C01894=67.036,-67.036,18.916,160.1256,-19.8741,0.0000
C01895=63.169,-70.689,18.914,159.1053,-18.7979,0.0000
C01896=59.448,-73.859,18.917,158.5547,-18.0191,0.0000
C01897=56.048,-76.685,18.976,160.0045,-17.9572,0.0000
C01898=53.950,-78.738,19.120,165.3862,-17.8366,0.0000
C01899=52.755,-80.388,19.309,171.7434,-14.7955,0.0000
C01900=51.961,-81.931,19.493,175.4363,-10.0997,0.0000
C01901=51.163,-83.502,19.627,176.4604,-6.1368,0.0000
C01902=49.917,-85.194,19.692,177.1673,-3.1412,0.0000
C01903=47.874,-87.106,19.726,178.6253,-1.1228,0.0000
C01904=45.272,-88.975,19.753,179.7684,-0.1462,0.0000
C01905=42.449,-90.515,19.780,179.9313,-0.0331,0.0000
C01906=39.659,-91.796,19.798,179.9923,-0.0034,0.0000
C01907=36.867,-92.953,19.798,179.9922,-0.0031,0.0000
C01908=33.988,-94.020,19.780,179.9280,-0.0252,0.0000
C01909=30.903,-94.927,19.753,179.7329,-0.0604,0.0000
C01910=27.741,-95.446,19.726,178.2343,-0.1783,0.0000
C01911=24.945,-95.538,19.692,175.7796,0.2187,0.0000
C01912=22.867,-95.222,19.627,173.1704,1.8493,0.0000
C01913=21.192,-94.676,19.493,169.6633,3.9762,0.0000
C01914=19.540,-94.146,19.309,163.8609,4.8105,0.0000
C01915=17.528,-93.824,19.120,157.6135,2.4711,0.0000
C01916=14.592,-93.857,18.976,154.0583,-1.6112,0.0000
C01917=10.190,-94.262,18.917,153.0799,-2.7339,0.0000
C01918=5.317,-94.652,18.914,152.9496,-1.6759,0.0000
C01919=0.000,-94.804,18.916,152.9230,0.0002,0.0000
C01920=0.000,-94.804,18.916,152.9230,0.0002,0.0000
C01921=-5.317,-94.652,18.914,152.9496,1.6756,0.0000
C01922=-10.190,-94.262,18.917,153.0799,2.7335,0.0000
C01923=-14.592,-93.857,18.976,154.0584,1.6115,0.0000
C01924=-17.528,-93.824,19.120,157.6135,-2.4711,0.0000
C01925=-19.540,-94.146,19.309,163.8609,-4.8105,0.0000
C01926=-21.192,-94.676,19.493,169.6633,-3.9762,0.0000
C01927=-22.867,-95.222,19.627,173.1704,-1.8493,0.0000
C01928=-24.945,-95.538,19.692,175.7796,-0.2187,0.0000
C01929=-27.741,-95.446,19.726,178.2343,0.1783,0.0000
C01930=-30.903,-94.927,19.753,179.7329,0.0604,0.0000
C01931=-33.988,-94.020,19.780,179.9280,0.0252,0.0000
C01932=-36.867,-92.953,19.798,179.9922,0.0031,0.0000
C01933=-39.659,-91.796,19.798,179.9923,0.0034,0.0000
C01934=-42.449,-90.515,19.780,179.9313,0.0331,0.0000
C01935=-45.272,-88.975,19.753,179.7684,0.1462,0.0000
C01936=-47.874,-87.106,19.726,178.6253,1.1228,0.0000
C01937=-49.917,-85.194,19.692,177.1673,3.1412,0.0000
C01938=-51.163,-83.502,19.627,176.4604,6.1368,0.0000
C01939=-51.961,-81.931,19.493,175.4363,10.0997,0.0000
C01940=-52.755,-80.388,19.309,171.7434,14.7955,0.0000
C01941=-53.950,-78.738,19.120,165.3862,17.8366,0.0000
C01942=-56.048,-76.685,18.976,160.0047,17.9574,0.0000
C01943=-59.448,-73.859,18.917,158.5544,18.0188,0.0000
C01944=-63.169,-70.689,18.914,159.1051,18.7977,0.0000
C01945=-67.036,-67.036,18.916,160.1259,19.8744,0.0000
C01946=-70.689,-63.169,18.914,161.2021,20.8947,0.0000
C01947=-73.859,-59.448,18.917,161.9809,21.4453,0.0000
C01948=-76.685,-56.048,18.976,162.0428,19.9955,0.0000
C01949=-78.738,-53.950,19.120,162.1634,14.6138,0.0000
C01950=-80.388,-52.755,19.309,165.2045,8.2566,0.0000
C01951=-81.931,-51.961,19.493,169.9003,4.5637,0.0000
C01952=-83.502,-51.163,19.627,173.8632,3.5396,0.0000
C01953=-85.194,-49.917,19.692,176.8588,2.8327,0.0000
C01954=-87.106,-47.874,19.726,178.8772,1.3747,0.0000
C01955=-88.975,-45.272,19.753,179.8538,0.2316,0.0000
C01956=-90.515,-42.449,19.780,179.9669,0.0687,0.0000
C01957=-91.796,-39.659,19.798,179.9966,0.0077,0.0000
C01958=-92.953,-36.867,19.798,179.9969,0.0078,0.0000
C01959=-94.020,-33.988,19.780,179.9748,0.0720,0.0000
C01960=-94.927,-30.903,19.753,179.9396,0.2671,0.0000
C01961=-95.446,-27.741,19.726,179.8217,1.7657,0.0000
C01962=-95.538,-24.945,19.692,-179.7813,4.2204,0.0000
C01963=-95.222,-22.867,19.627,-178.1507,6.8296,0.0000
C01964=-94.676,-21.192,19.493,-176.0238,10.3367,0.0000
C01965=-94.146,-19.540,19.309,-175.1895,16.1391,0.0000
C01966=-93.824,-17.528,19.120,-177.5289,22.3865,0.0000
C01967=-93.857,-14.592,18.976,178.3888,25.9417,0.0000
C01968=-94.262,-10.190,18.917,177.2661,26.9201,0.0000
C01969=-94.652,-5.317,18.914,178.3241,27.0504,0.0000
C01970=-94.804,0.000,18.916,-179.9998,27.0770,0.0000
C01971=-94.652,5.317,18.914,-178.3244,27.0504,0.0000
C01972=-94.262,10.190,18.917,-177.2665,26.9201,0.0000
C01973=-93.857,14.592,18.976,-178.3885,25.9416,0.0000
C01974=-93.824,17.528,19.120,177.5289,22.3865,0.0000
C01975=-94.146,19.540,19.309,175.1895,16.1391,0.0000
C01976=-94.676,21.192,19.493,176.0238,10.3367,0.0000
C01977=-95.222,22.867,19.627,178.1507,6.8296,0.0000
C01978=-95.538,24.945,19.692,179.7813,4.2204,0.0000
C01979=-95.446,27.741,19.726,-179.8217,1.7657,0.0000
C01980=-94.927,30.903,19.753,-179.9396,0.2671,0.0000
C01981=-94.020,33.988,19.780,-179.9748,0.0720,0.0000
C01982=-92.953,36.867,19.798,-179.9969,0.0078,0.0000
C01983=-91.796,39.659,19.798,-179.9966,0.0077,0.0000
C01984=-90.515,42.449,19.780,-179.9669,0.0687,0.0000
C01985=-88.975,45.272,19.753,-179.8538,0.2316,0.0000
C01986=-87.106,47.874,19.726,-178.8772,1.3747,0.0000
C01987=-85.194,49.917,19.692,-176.8588,2.8327,0.0000
C01988=-83.502,51.163,19.627,-173.8632,3.5396,0.0000
C01989=-81.931,51.961,19.493,-169.9003,4.5637,0.0000
C01990=-80.388,52.755,19.309,-165.2045,8.2566,0.0000
C01991=-78.738,53.950,19.120,-162.1634,14.6138,0.0000
C01992=-76.685,56.048,18.976,-162.0426,19.9953,0.0000
C01993=-73.859,59.448,18.917,-161.9812,21.4456,0.0000
C01994=-70.689,63.169,18.914,-161.2023,20.8949,0.0000
C01995=-67.036,67.036,18.916,-160.1256,19.8741,0.0000
C01996=-63.169,70.689,18.914,-159.1053,18.7979,0.0000
C01997=-59.448,73.859,18.917,-158.5547,18.0191,0.0000
C01998=-56.048,76.685,18.976,-160.0045,17.9572,0.0000
C01999=-53.950,78.738,19.120,-165.3862,17.8366,0.0000
///TOOL 0
///POSTYPE ANGLE
///ANGLE
EC00000=0.0000,0.0000
EC00001=0.0000,0.0000
EC00002=3.3204,0.0000
EC00003=6.3084,0.0000
EC00004=8.9540,0.0000
EC00005=10.7765,0.0000
EC00006=12.0369,0.0000
EC00007=13.0576,0.0000
EC00008=14.0938,0.0000
EC00009=15.3967,0.0000
EC00010=17.0065,0.0000
EC00011=18.7198,0.0000
EC00012=20.3278,0.0000
EC00013=21.7902,0.0000
EC00014=23.2098,0.0000
EC00015=24.6724,0.0000
EC00016=26.2801,0.0000
EC00017=27.9935,0.0000
EC00018=29.6039,0.0000
EC00019=30.9060,0.0000
EC00020=31.9421,0.0000
EC00021=32.9632,0.0000
EC00022=34.2234,0.0000
EC00023=36.0464,0.0000
EC00024=38.6909,0.0000
EC00025=41.6796,0.0000
EC00026=45.0000,0.0000
EC00027=48.3204,0.0000
EC00028=51.3091,0.0000
EC00029=53.9536,0.0000
EC00030=55.7766,0.0000
EC00031=57.0368,0.0000
EC00032=58.0579,0.0000
EC00033=59.0940,0.0000
EC00034=60.3961,0.0000
EC00035=62.0065,0.0000
EC00036=63.7199,0.0000
EC00037=65.3276,0.0000
EC00038=66.7902,0.0000
EC00039=68.2098,0.0000
EC00040=69.6722,0.0000
EC00041=71.2802,0.0000
EC00042=72.9935,0.0000
EC00043=74.6033,0.0000
EC00044=75.9062,0.0000
EC00045=76.9424,0.0000
EC00046=77.9631,0.0000
EC00047=79.2235,0.0000
EC00048=81.0460,0.0000
EC00049=83.6916,0.0000
EC00050=86.6796,0.0000
EC00051=90.0000,0.0000
EC00052=93.3204,0.0000
EC00053=96.3084,0.0000
EC00054=98.9540,0.0000
EC00055=100.7765,0.0000
EC00056=102.0369,0.0000
EC00057=103.0576,0.0000
EC00058=104.0938,0.0000
EC00059=105.3967,0.0000
EC00060=107.0065,0.0000
EC00061=108.7198,0.0000
EC00062=110.3278,0.0000
EC00063=111.7902,0.0000
EC00064=113.2098,0.0000
EC00065=114.6724,0.0000
EC00066=116.2801,0.0000
EC00067=117.9935,0.0000
EC00068=119.6039,0.0000
EC00069=120.9060,0.0000
EC00070=121.9421,0.0000
EC00071=122.9632,0.0000
EC00072=124.2234,0.0000
EC00073=126.0464,0.0000
EC00074=128.6909,0.0000
EC00075=131.6796,0.0000
EC00076=135.0000,0.0000
EC00077=138.3204,0.0000
EC00078=141.3091,0.0000
EC00079=143.9536,0.0000
EC00080=145.7766,0.0000
EC00081=147.0368,0.0000
EC00082=148.0579,0.0000
EC00083=149.0940,0.0000
EC00084=150.3961,0.0000
EC00085=152.0065,0.0000
EC00086=153.7199,0.0000
EC00087=155.3276,0.0000
EC00088=156.7902,0.0000
EC00089=158.2098,0.0000
EC00090=159.6722,0.0000
EC00091=161.2802,0.0000
EC00092=162.9935,0.0000
EC00093=164.6033,0.0000
EC00094=165.9062,0.0000
EC00095=166.9424,0.0000
EC00096=167.9631,0.0000
EC00097=169.2235,0.0000
EC00098=171.0460,0.0000
EC00099=173.6916,0.0000
EC00100=176.6796,0.0000
EC00101=180.0000,0.0000
EC00102=180.0000,0.0000
EC00103=-176.6796,0.0000
EC00104=-173.6916,0.0000
EC00105=-171.0460,0.0000
EC00106=-169.2235,0.0000
EC00107=-167.9631,0.0000
EC00108=-166.9424,0.0000
EC00109=-165.9062,0.0000
EC00110=-164.6033,0.0000
EC00111=-162.9935,0.0000
EC00112=-161.2802,0.0000
EC00113=-159.6722,0.0000
EC00114=-158.2098,0.0000
EC00115=-156.7902,0.0000
EC00116=-155.3276,0.0000
EC00117=-153.7199,0.0000
EC00118=-152.0065,0.0000
EC00119=-150.3961,0.0000
EC00120=-149.0940,0.0000
EC00121=-148.0579,0.0000
EC00122=-147.0368,0.0000
EC00123=-145.7766,0.0000
EC00124=-143.9536,0.0000
EC00125=-141.3091,0.0000
EC00126=-138.3204,0.0000
EC00127=-135.0000,0.0000
EC00128=-131.6796,0.0000
EC00129=-128.6909,0.0000
EC00130=-126.0464,0.0000
EC00131=-124.2234,0.0000
EC00132=-122.9632,0.0000
EC00133=-121.9421,0.0000
EC00134=-120.9060,0.0000
EC00135=-119.6039,0.0000
EC00136=-117.9935,0.0000
EC00137=-116.2801,0.0000
EC00138=-114.6724,0.0000
EC00139=-113.2098,0.0000
EC00140=-111.7902,0.0000
EC00141=-110.3278,0.0000
EC00142=-108.7198,0.0000
EC00143=-107.0065,0.0000
EC00144=-105.3967,0.0000
EC00145=-104.0938,0.0000
EC00146=-103.0576,0.0000
EC00147=-102.0369,0.0000
EC00148=-100.7765,0.0000
EC00149=-98.9540,0.0000
EC00150=-96.3084,0.0000
EC00151=-93.3204,0.0000
EC00152=-90.0000,0.0000
EC00153=-86.6796,0.0000
EC00154=-83.6916,0.0000
EC00155=-81.0460,0.0000
EC00156=-79.2235,0.0000
EC00157=-77.9631,0.0000
EC00158=-76.9424,0.0000
EC00159=-75.9062,0.0000
EC00160=-74.6033,0.0000
EC00161=-72.9935,0.0000
EC00162=-71.2802,0.0000
EC00163=-69.6722,0.0000
EC00164=-68.2098,0.0000
EC00165=-66.7902,0.0000
EC00166=-65.3276,0.0000
EC00167=-63.7199,0.0000
EC00168=-62.0065,0.0000
EC00169=-60.3961,0.0000
EC00170=-59.0940,0.0000
EC00171=-58.0579,0.0000
EC00172=-57.0368,0.0000
EC00173=-55.7766,0.0000
EC00174=-53.9536,0.0000
EC00175=-51.3091,0.0000
EC00176=-48.3204,0.0000
EC00177=-45.0000,0.0000
EC00178=-41.6796,0.0000
EC00179=-38.6909,0.0000
EC00180=-36.0464,0.0000
EC00181=-34.2234,0.0000
EC00182=-32.9632,0.0000
EC00183=-31.9421,0.0000
EC00184=-30.9060,0.0000
EC00185=-29.6039,0.0000
EC00186=-27.9935,0.0000
EC00187=-26.2801,0.0000
EC00188=-24.6724,0.0000
EC00189=-23.2098,0.0000
EC00190=-21.7902,0.0000
EC00191=-20.3278,0.0000
EC00192=-18.7198,0.0000
EC00193=-17.0065,0.0000
EC00194=-15.3967,0.0000
EC00195=-14.0938,0.0000
EC00196=-13.0576,0.0000
EC00197=-12.0369,0.0000
EC00198=-10.7765,0.0000
EC00199=-8.9540,0.0000
EC00200=-6.3084,0.0000
EC00201=-3.3204,0.0000
EC00202=0.0000,0.0000
EC00203=0.0000,0.0000
EC00204=3.3190,0.0000
EC00205=6.3064,0.0000
EC00206=8.9521,0.0000
EC00207=10.7740,0.0000
EC00208=12.0325,0.0000
EC00209=13.0515,0.0000
EC00210=14.0856,0.0000
EC00211=15.3858,0.0000
EC00212=16.9948,0.0000
EC00213=18.7100,0.0000
EC00214=20.3211,0.0000
EC00215=21.7884,0.0000
EC00216=23.2118,0.0000
EC00217=24.6788,0.0000
EC00218=26.2904,0.0000
EC00219=28.0051,0.0000
EC00220=29.6142,0.0000
EC00221=30.9142,0.0000
EC00222=31.9485,0.0000
EC00223=32.9671,0.0000
EC00224=34.2260,0.0000
EC00225=36.0482,0.0000
EC00226=38.6933,0.0000
EC00227=41.6811,0.0000
EC00228=45.0000,0.0000
EC00229=48.3189,0.0000
EC00230=51.3067,0.0000
EC00231=53.9518,0.0000
EC00232=55.7740,0.0000
EC00233=57.0329,0.0000
EC00234=58.0515,0.0000
EC00235=59.0858,0.0000
EC00236=60.3858,0.0000
EC00237=61.9949,0.0000
EC00238=63.7096,0.0000
EC00239=65.3212,0.0000
EC00240=66.7882,0.0000
EC00241=68.2116,0.0000
EC00242=69.6789,0.0000
EC00243=71.2900,0.0000
EC00244=73.0052,0.0000
EC00245=74.6142,0.0000
EC00246=75.9144,0.0000
EC00247=76.9485,0.0000
EC00248=77.9675,0.0000
EC00249=79.2260,0.0000
EC00250=81.0479,0.0000
EC00251=83.6936,0.0000
EC00252=86.6810,0.0000
EC00253=90.0000,0.0000
EC00254=93.3190,0.0000
EC00255=96.3064,0.0000
EC00256=98.9521,0.0000
EC00257=100.7740,0.0000
EC00258=102.0325,0.0000
EC00259=103.0515,0.0000
EC00260=104.0856,0.0000
EC00261=105.3858,0.0000
EC00262=106.9948,0.0000
EC00263=108.7100,0.0000
EC00264=110.3211,0.0000
EC00265=111.7884,0.0000
EC00266=113.2118,0.0000
EC00267=114.6788,0.0000
EC00268=116.2904,0.0000
EC00269=118.0051,0.0000
EC00270=119.6142,0.0000
EC00271=120.9142,0.0000
EC00272=121.9485,0.0000
EC00273=122.9671,0.0000
EC00274=124.2260,0.0000
EC00275=126.0482,0.0000
EC00276=128.6933,0.0000
EC00277=131.6811,0.0000
EC00278=135.0000,0.0000
EC00279=138.3189,0.0000
EC00280=141.3067,0.0000
EC00281=143.9518,0.0000
EC00282=145.7740,0.0000
EC00283=147.0329,0.0000
EC00284=148.0515,0.0000
EC00285=149.0858,0.0000
EC00286=150.3858,0.0000
EC00287=151.9949,0.0000
EC00288=153.7096,0.0000
EC00289=155.3212,0.0000
EC00290=156.7882,0.0000
EC00291=158.2116,0.0000
EC00292=159.6789,0.0000
EC00293=161.2900,0.0000
EC00294=163.0052,0.0000
EC00295=164.6142,0.0000
EC00296=165.9144,0.0000
EC00297=166.9485,0.0000
EC00298=167.9675,0.0000
EC00299=169.2260,0.0000
EC00300=171.0479,0.0000
EC00301=173.6936,0.0000
EC00302=176.6810,0.0000
EC00303=180.0000,0.0000
EC00304=180.0000,0.0000
EC00305=-176.6810,0.0000
EC00306=-173.6936,0.0000
EC00307=-171.0479,0.0000
EC00308=-169.2260,0.0000
EC00309=-167.9675,0.0000
EC00310=-166.9485,0.0000
EC00311=-165.9144,0.0000
EC00312=-164.6142,0.0000
EC00313=-163.0052,0.0000
EC00314=-161.2900,0.0000
EC00315=-159.6789,0.0000
EC00316=-158.2116,0.0000
EC00317=-156.7882,0.0000
EC00318=-155.3212,0.0000
EC00319=-153.7096,0.0000
EC00320=-151.9949,0.0000
EC00321=-150.3858,0.0000
EC00322=-149.0858,0.0000
EC00323=-148.0515,0.0000
EC00324=-147.0329,0.0000
EC00325=-145.7740,0.0000
EC00326=-143.9518,0.0000
EC00327=-141.3067,0.0000
EC00328=-138.3189,0.0000
EC00329=-135.0000,0.0000
EC00330=-131.6811,0.0000
EC00331=-128.6933,0.0000
EC00332=-126.0482,0.0000
EC00333=-124.2260,0.0000
EC00334=-122.9671,0.0000
EC00335=-121.9485,0.0000
EC00336=-120.9142,0.0000
EC00337=-119.6142,0.0000
EC00338=-118.0051,0.0000
EC00339=-116.2904,0.0000
EC00340=-114.6788,0.0000
EC00341=-113.2118,0.0000
EC00342=-111.7884,0.0000
EC00343=-110.3211,0.0000
EC00344=-108.7100,0.0000
EC00345=-106.9948,0.0000
EC00346=-105.3858,0.0000
EC00347=-104.0856,0.0000
EC00348=-103.0515,0.0000
EC00349=-102.0325,0.0000
EC00350=-100.7740,0.0000
EC00351=-98.9521,0.0000
EC00352=-96.3064,0.0000
EC00353=-93.3190,0.0000
EC00354=-90.0000,0.0000
EC00355=-86.6810,0.0000
EC00356=-83.6936,0.0000
EC00357=-81.0479,0.0000
EC00358=-79.2260,0.0000
EC00359=-77.9675,0.0000
EC00360=-76.9485,0.0000
EC00361=-75.9144,0.0000
EC00362=-74.6142,0.0000
EC00363=-73.0052,0.0000
EC00364=-71.2900,0.0000
EC00365=-69.6789,0.0000
EC00366=-68.2116,0.0000
EC00367=-66.7882,0.0000
EC00368=-65.3212,0.0000
EC00369=-63.7096,0.0000
EC00370=-61.9949,0.0000
EC00371=-60.3858,0.0000
EC00372=-59.0858,0.0000
EC00373=-58.0515,0.0000
EC00374=-57.0329,0.0000
EC00375=-55.7740,0.0000
EC00376=-53.9518,0.0000
EC00377=-51.3067,0.0000
EC00378=-48.3189,0.0000
EC00379=-45.0000,0.0000
EC00380=-41.6811,0.0000
EC00381=-38.6933,0.0000
EC00382=-36.0482,0.0000
EC00383=-34.2260,0.0000
EC00384=-32.9671,0.0000
EC00385=-31.9485,0.0000
EC00386=-30.9142,0.0000
EC00387=-29.6142,0.0000
EC00388=-28.0051,0.0000
EC00389=-26.2904,0.0000
EC00390=-24.6788,0.0000
EC00391=-23.2118,0.0000
EC00392=-21.7884,0.0000
EC00393=-20.3211,0.0000
EC00394=-18.7100,0.0000
EC00395=-16.9948,0.0000
EC00396=-15.3858,0.0000
EC00397=-14.0856,0.0000
EC00398=-13.0515,0.0000
EC00399=-12.0325,0.0000
EC00400=-10.7740,0.0000
EC00401=-8.9521,0.0000
EC00402=-6.3064,0.0000
EC00403=-3.3190,0.0000
EC00404=0.0000,0.0000
EC00405=0.0000,0.0000
EC00406=3.3146,0.0000
EC00407=6.3008,0.0000
EC00408=8.9471,0.0000
EC00409=10.7659,0.0000
EC00410=12.0199,0.0000
EC00411=13.0335,0.0000
EC00412=14.0616,0.0000
EC00413=15.3544,0.0000
EC00414=16.9622,0.0000
EC00415=18.6812,0.0000
EC00416=20.3024,0.0000
EC00417=21.7817,0.0000
EC00418=23.2185,0.0000
EC00419=24.6975,0.0000
EC00420=26.3188,0.0000
EC00421=28.0383,0.0000
EC00422=29.6456,0.0000
EC00423=30.9386,0.0000
EC00424=31.9667,0.0000
EC00425=32.9801,0.0000
EC00426=34.2340,0.0000
EC00427=36.0529,0.0000
EC00428=38.6992,0.0000
EC00429=41.6856,0.0000
EC00430=45.0000,0.0000
EC00431=48.3144,0.0000
EC00432=51.3008,0.0000
EC00433=53.9471,0.0000
EC00434=55.7660,0.0000
EC00435=57.0199,0.0000
EC00436=58.0333,0.0000
EC00437=59.0614,0.0000
EC00438=60.3544,0.0000
EC00439=61.9617,0.0000
EC00440=63.6812,0.0000
EC00441=65.3025,0.0000
EC00442=66.7815,0.0000
EC00443=68.2183,0.0000
EC00444=69.6976,0.0000
EC00445=71.3188,0.0000
EC00446=73.0378,0.0000
EC00447=74.6456,0.0000
EC00448=75.9384,0.0000
EC00449=76.9665,0.0000
EC00450=77.9801,0.0000
EC00451=79.2341,0.0000
EC00452=81.0529,0.0000
EC00453=83.6992,0.0000
EC00454=86.6854,0.0000
EC00455=90.0000,0.0000
EC00456=93.3146,0.0000
EC00457=96.3008,0.0000
EC00458=98.9471,0.0000
EC00459=100.7659,0.0000
EC00460=102.0199,0.0000
EC00461=103.0335,0.0000
EC00462=104.0616,0.0000
EC00463=105.3544,0.0000
EC00464=106.9622,0.0000
EC00465=108.6812,0.0000
EC00466=110.3024,0.0000
EC00467=111.7817,0.0000
EC00468=113.2185,0.0000
EC00469=114.6975,0.0000
EC00470=116.3188,0.0000
EC00471=118.0383,0.0000
EC00472=119.6456,0.0000
EC00473=120.9386,0.0000
EC00474=121.9667,0.0000
EC00475=122.9801,0.0000
EC00476=124.2340,0.0000
EC00477=126.0529,0.0000
EC00478=128.6992,0.0000
EC00479=131.6856,0.0000
EC00480=135.0000,0.0000
EC00481=138.3144,0.0000
EC00482=141.3008,0.0000
EC00483=143.9471,0.0000
EC00484=145.7660,0.0000
EC00485=147.0199,0.0000
EC00486=148.0333,0.0000
EC00487=149.0614,0.0000
EC00488=150.3544,0.0000
EC00489=151.9617,0.0000
EC00490=153.6812,0.0000
EC00491=155.3025,0.0000
EC00492=156.7815,0.0000
EC00493=158.2183,0.0000
EC00494=159.6976,0.0000
EC00495=161.3188,0.0000
EC00496=163.0378,0.0000
EC00497=164.6456,0.0000
EC00498=165.9384,0.0000
EC00499=166.9665,0.0000
EC00500=167.9801,0.0000
EC00501=169.2341,0.0000
EC00502=171.0529,0.0000
EC00503=173.6992,0.0000
EC00504=176.6854,0.0000
EC00505=180.0000,0.0000
EC00506=180.0000,0.0000
EC00507=-176.6854,0.0000
EC00508=-173.6992,0.0000
EC00509=-171.0529,0.0000
EC00510=-169.2341,0.0000
EC00511=-167.9801,0.0000
EC00512=-166.9665,0.0000
EC00513=-165.9384,0.0000
EC00514=-164.6456,0.0000
EC00515=-163.0378,0.0000
EC00516=-161.3188,0.0000
EC00517=-159.6976,0.0000
EC00518=-158.2183,0.0000
EC00519=-156.7815,0.0000
EC00520=-155.3025,0.0000
EC00521=-153.6812,0.0000
EC00522=-151.9617,0.0000
EC00523=-150.3544,0.0000
EC00524=-149.0614,0.0000
EC00525=-148.0333,0.0000
EC00526=-147.0199,0.0000
EC00527=-145.7660,0.0000
EC00528=-143.9471,0.0000
EC00529=-141.3008,0.0000
EC00530=-138.3144,0.0000
EC00531=-135.0000,0.0000
EC00532=-131.6856,0.0000
EC00533=-128.6992,0.0000
EC00534=-126.0529,0.0000
EC00535=-124.2340,0.0000
EC00536=-122.9801,0.0000
EC00537=-121.9667,0.0000
EC00538=-120.9386,0.0000
EC00539=-119.6456,0.0000
EC00540=-118.0383,0.0000
EC00541=-116.3188,0.0000
EC00542=-114.6975,0.0000
EC00543=-113.2185,0.0000
EC00544=-111.7817,0.0000
EC00545=-110.3024,0.0000
EC00546=-108.6812,0.0000
EC00547=-106.9622,0.0000
EC00548=-105.3544,0.0000
EC00549=-104.0616,0.0000
EC00550=-103.0335,0.0000
EC00551=-102.0199,0.0000
EC00552=-100.7659,0.0000
EC00553=-98.9471,0.0000
EC00554=-96.3008,0.0000
EC00555=-93.3146,0.0000
EC00556=-90.0000,0.0000
EC00557=-86.6854,0.0000
EC00558=-83.6992,0.0000
EC00559=-81.0529,0.0000
EC00560=-79.2341,0.0000
EC00561=-77.9801,0.0000
EC00562=-76.9665,0.0000
EC00563=-75.9384,0.0000
EC00564=-74.6456,0.0000
EC00565=-73.0378,0.0000
EC00566=-71.3188,0.0000
EC00567=-69.6976,0.0000
EC00568=-68.2183,0.0000
EC00569=-66.7815,0.0000
EC00570=-65.3025,0.0000
EC00571=-63.6812,0.0000
EC00572=-61.9617,0.0000
EC00573=-60.3544,0.0000
EC00574=-59.0614,0.0000
EC00575=-58.0333,0.0000
EC00576=-57.0199,0.0000
EC00577=-55.7660,0.0000
EC00578=-53.9471,0.0000
EC00579=-51.3008,0.0000
EC00580=-48.3144,0.0000
EC00581=-45.0000,0.0000
EC00582=-41.6856,0.0000
EC00583=-38.6992,0.0000
EC00584=-36.0529,0.0000
EC00585=-34.2340,0.0000
EC00586=-32.9801,0.0000
EC00587=-31.9667,0.0000
EC00588=-30.9386,0.0000
EC00589=-29.6456,0.0000
EC00590=-28.0383,0.0000
EC00591=-26.3188,0.0000
EC00592=-24.6975,0.0000
EC00593=-23.2185,0.0000
EC00594=-21.7817,0.0000
EC00595=-20.3024,0.0000
EC00596=-18.6812,0.0000
EC00597=-16.9622,0.0000
EC00598=-15.3544,0.0000
EC00599=-14.0616,0.0000
EC00600=-13.0335,0.0000
EC00601=-12.0199,0.0000
EC00602=-10.7659,0.0000
EC00603=-8.9471,0.0000
EC00604=-6.3008,0.0000
EC00605=-3.3146,0.0000
EC00606=0.0000,0.0000
EC00607=0.0000,0.0000
EC00608=3.3073,0.0000
EC00609=6.2913,0.0000
EC00610=8.9391,0.0000
EC00611=10.7524,0.0000
EC00612=11.9986,0.0000
EC00613=13.0036,0.0000
EC00614=14.0220,0.0000
EC00615=15.3030,0.0000
EC00616=16.9082,0.0000
EC00617=18.6350,0.0000
EC00618=20.2716,0.0000
EC00619=21.7712,0.0000
EC00620=23.2288,0.0000
EC00621=24.7282,0.0000
EC00622=26.3649,0.0000
EC00623=28.0920,0.0000
EC00624=29.6973,0.0000
EC00625=30.9780,0.0000
EC00626=31.9962,0.0000
EC00627=33.0013,0.0000
EC00628=34.2478,0.0000
EC00629=36.0610,0.0000
EC00630=38.7088,0.0000
EC00631=41.6924,0.0000
EC00632=45.0000,0.0000
EC00633=48.3076,0.0000
EC00634=51.2912,0.0000
EC00635=53.9390,0.0000
EC00636=55.7522,0.0000
EC00637=56.9987,0.0000
EC00638=58.0038,0.0000
EC00639=59.0220,0.0000
EC00640=60.3027,0.0000
EC00641=61.9080,0.0000
EC00642=63.6351,0.0000
EC00643=65.2718,0.0000
EC00644=66.7712,0.0000
EC00645=68.2288,0.0000
EC00646=69.7284,0.0000
EC00647=71.3650,0.0000
EC00648=73.0918,0.0000
EC00649=74.6970,0.0000
EC00650=75.9780,0.0000
EC00651=76.9964,0.0000
EC00652=78.0014,0.0000
EC00653=79.2476,0.0000
EC00654=81.0609,0.0000
EC00655=83.7087,0.0000
EC00656=86.6927,0.0000
EC00657=90.0000,0.0000
EC00658=93.3073,0.0000
EC00659=96.2913,0.0000
EC00660=98.9391,0.0000
EC00661=100.7524,0.0000
EC00662=101.9986,0.0000
EC00663=103.0036,0.0000
EC00664=104.0220,0.0000
EC00665=105.3030,0.0000
EC00666=106.9082,0.0000
EC00667=108.6350,0.0000
EC00668=110.2716,0.0000
EC00669=111.7712,0.0000
EC00670=113.2288,0.0000
EC00671=114.7282,0.0000
EC00672=116.3649,0.0000
EC00673=118.0920,0.0000
EC00674=119.6973,0.0000
EC00675=120.9780,0.0000
EC00676=121.9962,0.0000
EC00677=123.0013,0.0000
EC00678=124.2478,0.0000
EC00679=126.0610,0.0000
EC00680=128.7088,0.0000
EC00681=131.6924,0.0000
EC00682=135.0000,0.0000
EC00683=138.3076,0.0000
EC00684=141.2912,0.0000
EC00685=143.9390,0.0000
EC00686=145.7522,0.0000
EC00687=146.9987,0.0000
EC00688=148.0038,0.0000
EC00689=149.0220,0.0000
EC00690=150.3027,0.0000
EC00691=151.9080,0.0000
EC00692=153.6351,0.0000
EC00693=155.2718,0.0000
EC00694=156.7712,0.0000
EC00695=158.2288,0.0000
EC00696=159.7284,0.0000
EC00697=161.3650,0.0000
EC00698=163.0918,0.0000
EC00699=164.6970,0.0000
EC00700=165.9780,0.0000
EC00701=166.9964,0.0000
EC00702=168.0014,0.0000
EC00703=169.2476,0.0000
EC00704=171.0609,0.0000
EC00705=173.7087,0.0000
EC00706=176.6927,0.0000
EC00707=180.0000,0.0000
EC00708=180.0000,0.0000
EC00709=-176.6927,0.0000
EC00710=-173.7087,0.0000
EC00711=-171.0609,0.0000
EC00712=-169.2476,0.0000
EC00713=-168.0014,0.0000
EC00714=-166.9964,0.0000
EC00715=-165.9780,0.0000
EC00716=-164.6970,0.0000
EC00717=-163.0918,0.0000
EC00718=-161.3650,0.0000
EC00719=-159.7284,0.0000
EC00720=-158.2288,0.0000
EC00721=-156.7712,0.0000
EC00722=-155.2718,0.0000
EC00723=-153.6351,0.0000
EC00724=-151.9080,0.0000
EC00725=-150.3027,0.0000
EC00726=-149.0220,0.0000
EC00727=-148.0038,0.0000
EC00728=-146.9987,0.0000
EC00729=-145.7522,0.0000
EC00730=-143.9390,0.0000
EC00731=-141.2912,0.0000
EC00732=-138.3076,0.0000
EC00733=-135.0000,0.0000
EC00734=-131.6924,0.0000
EC00735=-128.7088,0.0000
EC00736=-126.0610,0.0000
EC00737=-124.2478,0.0000
EC00738=-123.0013,0.0000
EC00739=-121.9962,0.0000
EC00740=-120.9780,0.0000
EC00741=-119.6973,0.0000
EC00742=-118.0920,0.0000
EC00743=-116.3649,0.0000
EC00744=-114.7282,0.0000
EC00745=-113.2288,0.0000
EC00746=-111.7712,0.0000
EC00747=-110.2716,0.0000
EC00748=-108.6350,0.0000
EC00749=-106.9082,0.0000
EC00750=-105.3030,0.0000
EC00751=-104.0220,0.0000
EC00752=-103.0036,0.0000
EC00753=-101.9986,0.0000
EC00754=-100.7524,0.0000
EC00755=-98.9391,0.0000
EC00756=-96.2913,0.0000
EC00757=-93.3073,0.0000
EC00758=-90.0000,0.0000
EC00759=-86.6927,0.0000
EC00760=-83.7087,0.0000
EC00761=-81.0609,0.0000
EC00762=-79.2476,0.0000
EC00763=-78.0014,0.0000
EC00764=-76.9964,0.0000
EC00765=-75.9780,0.0000
EC00766=-74.6970,0.0000
EC00767=-73.0918,0.0000
EC00768=-71.3650,0.0000
EC00769=-69.7284,0.0000
EC00770=-68.2288,0.0000
EC00771=-66.7712,0.0000
EC00772=-65.2718,0.0000
EC00773=-63.6351,0.0000
EC00774=-61.9080,0.0000
EC00775=-60.3027,0.0000
EC00776=-59.0220,0.0000
EC00777=-58.0038,0.0000
EC00778=-56.9987,0.0000
EC00779=-55.7522,0.0000
EC00780=-53.9390,0.0000
EC00781=-51.2912,0.0000
EC00782=-48.3076,0.0000
EC00783=-45.0000,0.0000
EC00784=-41.6924,0.0000
EC00785=-38.7088,0.0000
EC00786=-36.0610,0.0000
EC00787=-34.2478,0.0000
EC00788=-33.0013,0.0000
EC00789=-31.9962,0.0000
EC00790=-30.9780,0.0000
EC00791=-29.6973,0.0000
EC00792=-28.0920,0.0000
EC00793=-26.3649,0.0000
EC00794=-24.7282,0.0000
EC00795=-23.2288,0.0000
EC00796=-21.7712,0.0000
EC00797=-20.2716,0.0000
EC00798=-18.6350,0.0000
EC00799=-16.9082,0.0000
EC00800=-15.3030,0.0000
EC00801=-14.0220,0.0000
EC00802=-13.0036,0.0000
EC00803=-11.9986,0.0000
EC00804=-10.7524,0.0000
EC00805=-8.9391,0.0000
EC00806=-6.2913,0.0000
EC00807=-3.3073,0.0000
EC00808=0.0000,0.0000
EC00809=0.0000,0.0000
EC00810=3.2974,0.0000
EC00811=6.2783,0.0000
EC00812=8.9284,0.0000
EC00813=10.7347,0.0000
EC00814=11.9700,0.0000
EC00815=12.9633,0.0000
EC00816=13.9678,0.0000
EC00817=15.2327,0.0000
EC00818=16.8342,0.0000
EC00819=18.5716,0.0000
EC00820=20.2300,0.0000
EC00821=21.7565,0.0000
EC00822=23.2431,0.0000
EC00823=24.7700,0.0000
EC00824=26.4284,0.0000
EC00825=28.1658,0.0000
EC00826=29.7669,0.0000
EC00827=31.0323,0.0000
EC00828=32.0364,0.0000
EC00829=33.0299,0.0000
EC00830=34.2655,0.0000
EC00831=36.0719,0.0000
EC00832=38.7215,0.0000
EC00833=41.7023,0.0000
EC00834=45.0000,0.0000
EC00835=48.2977,0.0000
EC00836=51.2785,0.0000
EC00837=53.9281,0.0000
EC00838=55.7345,0.0000
EC00839=56.9701,0.0000
EC00840=57.9636,0.0000
EC00841=58.9677,0.0000
EC00842=60.2331,0.0000
EC00843=61.8342,0.0000
EC00844=63.5716,0.0000
EC00845=65.2300,0.0000
EC00846=66.7569,0.0000
EC00847=68.2435,0.0000
EC00848=69.7700,0.0000
EC00849=71.4284,0.0000
EC00850=73.1658,0.0000
EC00851=74.7673,0.0000
EC00852=76.0322,0.0000
EC00853=77.0367,0.0000
EC00854=78.0300,0.0000
EC00855=79.2653,0.0000
EC00856=81.0716,0.0000
EC00857=83.7217,0.0000
EC00858=86.7026,0.0000
EC00859=90.0000,0.0000
EC00860=93.2974,0.0000
EC00861=96.2783,0.0000
EC00862=98.9284,0.0000
EC00863=100.7347,0.0000
EC00864=101.9700,0.0000
EC00865=102.9633,0.0000
EC00866=103.9678,0.0000
EC00867=105.2327,0.0000
EC00868=106.8342,0.0000
EC00869=108.5716,0.0000
EC00870=110.2300,0.0000
EC00871=111.7565,0.0000
EC00872=113.2431,0.0000
EC00873=114.7700,0.0000
EC00874=116.4284,0.0000
EC00875=118.1658,0.0000
EC00876=119.7669,0.0000
EC00877=121.0323,0.0000
EC00878=122.0364,0.0000
EC00879=123.0299,0.0000
EC00880=124.2655,0.0000
EC00881=126.0719,0.0000
EC00882=128.7215,0.0000
EC00883=131.7023,0.0000
EC00884=135.0000,0.0000
EC00885=138.2977,0.0000
EC00886=141.2785,0.0000
EC00887=143.9281,0.0000
EC00888=145.7345,0.0000
EC00889=146.9701,0.0000
EC00890=147.9636,0.0000
EC00891=148.9677,0.0000
EC00892=150.2331,0.0000
EC00893=151.8342,0.0000
EC00894=153.5716,0.0000
EC00895=155.2300,0.0000
EC00896=156.7569,0.0000
EC00897=158.2435,0.0000
EC00898=159.7700,0.0000
EC00899=161.4284,0.0000
EC00900=163.1658,0.0000
EC00901=164.7673,0.0000
EC00902=166.0322,0.0000
EC00903=167.0367,0.0000
EC00904=168.0300,0.0000
EC00905=169.2653,0.0000
EC00906=171.0716,0.0000
EC00907=173.7217,0.0000
EC00908=176.7026,0.0000
EC00909=180.0000,0.0000
EC00910=180.0000,0.0000
EC00911=-176.7026,0.0000
EC00912=-173.7217,0.0000
EC00913=-171.0716,0.0000
EC00914=-169.2653,0.0000
EC00915=-168.0300,0.0000
EC00916=-167.0367,0.0000
EC00917=-166.0322,0.0000
EC00918=-164.7673,0.0000
EC00919=-163.1658,0.0000
EC00920=-161.4284,0.0000
EC00921=-159.7700,0.0000
EC00922=-158.2435,0.0000
EC00923=-156.7569,0.0000
EC00924=-155.2300,0.0000
EC00925=-153.5716,0.0000
EC00926=-151.8342,0.0000
EC00927=-150.2331,0.0000
EC00928=-148.9677,0.0000
EC00929=-147.9636,0.0000
EC00930=-146.9701,0.0000
EC00931=-145.7345,0.0000
EC00932=-143.9281,0.0000
EC00933=-141.2785,0.0000
EC00934=-138.2977,0.0000
EC00935=-135.0000,0.0000
EC00936=-131.7023,0.0000
EC00937=-128.7215,0.0000
EC00938=-126.0719,0.0000
EC00939=-124.2655,0.0000
EC00940=-123.0299,0.0000
EC00941=-122.0364,0.0000
EC00942=-121.0323,0.0000
EC00943=-119.7669,0.0000
EC00944=-118.1658,0.0000
EC00945=-116.4284,0.0000
EC00946=-114.7700,0.0000
EC00947=-113.2431,0.0000
EC00948=-111.7565,0.0000
EC00949=-110.2300,0.0000
EC00950=-108.5716,0.0000
EC00951=-106.8342,0.0000
EC00952=-105.2327,0.0000
EC00953=-103.9678,0.0000
EC00954=-102.9633,0.0000
EC00955=-101.9700,0.0000
EC00956=-100.7347,0.0000
EC00957=-98.9284,0.0000
EC00958=-96.2783,0.0000
EC00959=-93.2974,0.0000
EC00960=-90.0000,0.0000
EC00961=-86.7026,0.0000
EC00962=-83.7217,0.0000
EC00963=-81.0716,0.0000
EC00964=-79.2653,0.0000
EC00965=-78.0300,0.0000
EC00966=-77.0367,0.0000
EC00967=-76.0322,0.0000
EC00968=-74.7673,0.0000
EC00969=-73.1658,0.0000
EC00970=-71.4284,0.0000
EC00971=-69.7700,0.0000
EC00972=-68.2435,0.0000
EC00973=-66.7569,0.0000
EC00974=-65.2300,0.0000
EC00975=-63.5716,0.0000
EC00976=-61.8342,0.0000
EC00977=-60.2331,0.0000
EC00978=-58.9677,0.0000
EC00979=-57.9636,0.0000
EC00980=-56.9701,0.0000
EC00981=-55.7345,0.0000
EC00982=-53.9281,0.0000
EC00983=-51.2785,0.0000
EC00984=-48.2977,0.0000
EC00985=-45.0000,0.0000
EC00986=-41.7023,0.0000
EC00987=-38.7215,0.0000
EC00988=-36.0719,0.0000
EC00989=-34.2655,0.0000
EC00990=-33.0299,0.0000
EC00991=-32.0364,0.0000
EC00992=-31.0323,0.0000
EC00993=-29.7669,0.0000
EC00994=-28.1658,0.0000
EC00995=-26.4284,0.0000
EC00996=-24.7700,0.0000
EC00997=-23.2431,0.0000
EC00998=-21.7565,0.0000
EC00999=-20.2300,0.0000
EC01000=-18.5716,0.0000
EC01001=-16.8342,0.0000
EC01002=-15.2327,0.0000
EC01003=-13.9678,0.0000
EC01004=-12.9633,0.0000
EC01005=-11.9700,0.0000
EC01006=-10.7347,0.0000
EC01007=-8.9284,0.0000
EC01008=-6.2783,0.0000
EC01009=-3.2974,0.0000
EC01010=0.0000,0.0000
EC01011=0.0000,0.0000
EC01012=3.2854,0.0000
EC01013=6.2621,0.0000
EC01014=8.9150,0.0000
EC01015=10.7121,0.0000
EC01016=11.9342,0.0000
EC01017=12.9128,0.0000
EC01018=13.8997,0.0000
EC01019=15.1448,0.0000
EC01020=16.7421,0.0000
EC01021=18.4921,0.0000
EC01022=20.1777,0.0000
EC01023=21.7387,0.0000
EC01024=23.2613,0.0000
EC01025=24.8225,0.0000
EC01026=26.5076,0.0000
EC01027=28.2578,0.0000
EC01028=29.8549,0.0000
EC01029=31.1001,0.0000
EC01030=32.0874,0.0000
EC01031=33.0661,0.0000
EC01032=34.2883,0.0000
EC01033=36.0850,0.0000
EC01034=38.7375,0.0000
EC01035=41.7146,0.0000
EC01036=45.0000,0.0000
EC01037=48.2854,0.0000
EC01038=51.2625,0.0000
EC01039=53.9150,0.0000
EC01040=55.7117,0.0000
EC01041=56.9339,0.0000
EC01042=57.9126,0.0000
EC01043=58.8999,0.0000
EC01044=60.1451,0.0000
EC01045=61.7422,0.0000
EC01046=63.4924,0.0000
EC01047=65.1775,0.0000
EC01048=66.7387,0.0000
EC01049=68.2613,0.0000
EC01050=69.8223,0.0000
EC01051=71.5079,0.0000
EC01052=73.2579,0.0000
EC01053=74.8552,0.0000
EC01054=76.1003,0.0000
EC01055=77.0872,0.0000
EC01056=78.0658,0.0000
EC01057=79.2879,0.0000
EC01058=81.0850,0.0000
EC01059=83.7379,0.0000
EC01060=86.7146,0.0000
EC01061=90.0000,0.0000
EC01062=93.2854,0.0000
EC01063=96.2621,0.0000
EC01064=98.9150,0.0000
EC01065=100.7121,0.0000
EC01066=101.9342,0.0000
EC01067=102.9128,0.0000
EC01068=103.8997,0.0000
EC01069=105.1448,0.0000
EC01070=106.7421,0.0000
EC01071=108.4921,0.0000
EC01072=110.1777,0.0000
EC01073=111.7387,0.0000
EC01074=113.2613,0.0000
EC01075=114.8225,0.0000
EC01076=116.5076,0.0000
EC01077=118.2578,0.0000
EC01078=119.8549,0.0000
EC01079=121.1001,0.0000
EC01080=122.0874,0.0000
EC01081=123.0661,0.0000
EC01082=124.2883,0.0000
EC01083=126.0850,0.0000
EC01084=128.7375,0.0000
EC01085=131.7146,0.0000
EC01086=135.0000,0.0000
EC01087=138.2854,0.0000
EC01088=141.2625,0.0000
EC01089=143.9150,0.0000
EC01090=145.7117,0.0000
EC01091=146.9339,0.0000
EC01092=147.9126,0.0000
EC01093=148.8999,0.0000
EC01094=150.1451,0.0000
EC01095=151.7422,0.0000
EC01096=153.4924,0.0000
EC01097=155.1775,0.0000
EC01098=156.7387,0.0000
EC01099=158.2613,0.0000
EC01100=159.8223,0.0000
EC01101=161.5079,0.0000
EC01102=163.2579,0.0000
EC01103=164.8552,0.0000
EC01104=166.1003,0.0000
EC01105=167.0872,0.0000
EC01106=168.0658,0.0000
EC01107=169.2879,0.0000
EC01108=171.0850,0.0000
EC01109=173.7379,0.0000
EC01110=176.7146,0.0000
EC01111=180.0000,0.0000
EC01112=180.0000,0.0000
EC01113=-176.7146,0.0000
EC01114=-173.7379,0.0000
EC01115=-171.0850,0.0000
EC01116=-169.2879,0.0000
EC01117=-168.0658,0.0000
EC01118=-167.0872,0.0000
EC01119=-166.1003,0.0000
EC01120=-164.8552,0.0000
EC01121=-163.2579,0.0000
EC01122=-161.5079,0.0000
EC01123=-159.8223,0.0000
EC01124=-158.2613,0.0000
EC01125=-156.7387,0.0000
EC01126=-155.1775,0.0000
EC01127=-153.4924,0.0000
EC01128=-151.7422,0.0000
EC01129=-150.1451,0.0000
EC01130=-148.8999,0.0000
EC01131=-147.9126,0.0000
EC01132=-146.9339,0.0000
EC01133=-145.7117,0.0000
EC01134=-143.9150,0.0000
EC01135=-141.2625,0.0000
EC01136=-138.2854,0.0000
EC01137=-135.0000,0.0000
EC01138=-131.7146,0.0000
EC01139=-128.7375,0.0000
EC01140=-126.0850,0.0000
EC01141=-124.2883,0.0000
EC01142=-123.0661,0.0000
EC01143=-122.0874,0.0000
EC01144=-121.1001,0.0000
EC01145=-119.8549,0.0000
EC01146=-118.2578,0.0000
EC01147=-116.5076,0.0000
EC01148=-114.8225,0.0000
EC01149=-113.2613,0.0000
EC01150=-111.7387,0.0000
EC01151=-110.1777,0.0000
EC01152=-108.4921,0.0000
EC01153=-106.7421,0.0000
EC01154=-105.1448,0.0000
EC01155=-103.8997,0.0000
EC01156=-102.9128,0.0000
EC01157=-101.9342,0.0000
EC01158=-100.7121,0.0000
EC01159=-98.9150,0.0000
EC01160=-96.2621,0.0000
EC01161=-93.2854,0.0000
EC01162=-90.0000,0.0000
EC01163=-86.7146,0.0000
EC01164=-83.7379,0.0000
EC01165=-81.0850,0.0000
EC01166=-79.2879,0.0000
EC01167=-78.0658,0.0000
EC01168=-77.0872,0.0000
EC01169=-76.1003,0.0000
EC01170=-74.8552,0.0000
EC01171=-73.2579,0.0000
EC01172=-71.5079,0.0000
EC01173=-69.8223,0.0000
EC01174=-68.2613,0.0000
EC01175=-66.7387,0.0000
EC01176=-65.1775,0.0000
EC01177=-63.4924,0.0000
EC01178=-61.7422,0.0000
EC01179=-60.1451,0.0000
EC01180=-58.8999,0.0000
EC01181=-57.9126,0.0000
EC01182=-56.9339,0.0000
EC01183=-55.7117,0.0000
EC01184=-53.9150,0.0000
EC01185=-51.2625,0.0000
EC01186=-48.2854,0.0000
EC01187=-45.0000,0.0000
EC01188=-41.7146,0.0000
EC01189=-38.7375,0.0000
EC01190=-36.0850,0.0000
EC01191=-34.2883,0.0000
EC01192=-33.0661,0.0000
EC01193=-32.0874,0.0000
EC01194=-31.1001,0.0000
EC01195=-29.8549,0.0000
EC01196=-28.2578,0.0000
EC01197=-26.5076,0.0000
EC01198=-24.8225,0.0000
EC01199=-23.2613,0.0000
EC01200=-21.7387,0.0000
EC01201=-20.1777,0.0000
EC01202=-18.4921,0.0000
EC01203=-16.7421,0.0000
EC01204=-15.1448,0.0000
EC01205=-13.8997,0.0000
EC01206=-12.9128,0.0000
EC01207=-11.9342,0.0000
EC01208=-10.7121,0.0000
EC01209=-8.9150,0.0000
EC01210=-6.2621,0.0000
EC01211=-3.2854,0.0000
EC01212=0.0000,0.0000
EC01213=0.0000,0.0000
EC01214=3.2709,0.0000
EC01215=6.2435,0.0000
EC01216=8.8988,0.0000
EC01217=10.6850,0.0000
EC01218=11.8912,0.0000
EC01219=12.8520,0.0000
EC01220=13.8189,0.0000
EC01221=15.0400,0.0000
EC01222=16.6318,0.0000
EC01223=18.3974,0.0000
EC01224=20.1155,0.0000
EC01225=21.7171,0.0000
EC01226=23.2826,0.0000
EC01227=24.8847,0.0000
EC01228=26.6022,0.0000
EC01229=28.3677,0.0000
EC01230=29.9600,0.0000
EC01231=31.1815,0.0000
EC01232=32.1481,0.0000
EC01233=33.1089,0.0000
EC01234=34.3149,0.0000
EC01235=36.1008,0.0000
EC01236=38.7567,0.0000
EC01237=41.7290,0.0000
EC01238=45.0000,0.0000
EC01239=48.2710,0.0000
EC01240=51.2433,0.0000
EC01241=53.8992,0.0000
EC01242=55.6851,0.0000
EC01243=56.8911,0.0000
EC01244=57.8519,0.0000
EC01245=58.8185,0.0000
EC01246=60.0400,0.0000
EC01247=61.6323,0.0000
EC01248=63.3978,0.0000
EC01249=65.1153,0.0000
EC01250=66.7174,0.0000
EC01251=68.2829,0.0000
EC01252=69.8845,0.0000
EC01253=71.6026,0.0000
EC01254=73.3682,0.0000
EC01255=74.9600,0.0000
EC01256=76.1811,0.0000
EC01257=77.1480,0.0000
EC01258=78.1088,0.0000
EC01259=79.3150,0.0000
EC01260=81.1012,0.0000
EC01261=83.7565,0.0000
EC01262=86.7291,0.0000
EC01263=90.0000,0.0000
EC01264=93.2709,0.0000
EC01265=96.2435,0.0000
EC01266=98.8988,0.0000
EC01267=100.6850,0.0000
EC01268=101.8912,0.0000
EC01269=102.8520,0.0000
EC01270=103.8189,0.0000
EC01271=105.0400,0.0000
EC01272=106.6318,0.0000
EC01273=108.3974,0.0000
EC01274=110.1155,0.0000
EC01275=111.7171,0.0000
EC01276=113.2826,0.0000
EC01277=114.8847,0.0000
EC01278=116.6022,0.0000
EC01279=118.3677,0.0000
EC01280=119.9600,0.0000
EC01281=121.1815,0.0000
EC01282=122.1481,0.0000
EC01283=123.1089,0.0000
EC01284=124.3149,0.0000
EC01285=126.1008,0.0000
EC01286=128.7567,0.0000
EC01287=131.7290,0.0000
EC01288=135.0000,0.0000
EC01289=138.2710,0.0000
EC01290=141.2433,0.0000
EC01291=143.8992,0.0000
EC01292=145.6851,0.0000
EC01293=146.8911,0.0000
EC01294=147.8519,0.0000
EC01295=148.8185,0.0000
EC01296=150.0400,0.0000
EC01297=151.6323,0.0000
EC01298=153.3978,0.0000
EC01299=155.1153,0.0000
EC01300=156.7174,0.0000
EC01301=158.2829,0.0000
EC01302=159.8845,0.0000
EC01303=161.6026,0.0000
EC01304=163.3682,0.0000
EC01305=164.9600,0.0000
EC01306=166.1811,0.0000
EC01307=167.1480,0.0000
EC01308=168.1088,0.0000
EC01309=169.3150,0.0000
EC01310=171.1012,0.0000
EC01311=173.7565,0.0000
EC01312=176.7291,0.0000
EC01313=180.0000,0.0000
EC01314=180.0000,0.0000
EC01315=-176.7291,0.0000
EC01316=-173.7565,0.0000
EC01317=-171.1012,0.0000
EC01318=-169.3150,0.0000
EC01319=-168.1088,0.0000
EC01320=-167.1480,0.0000
EC01321=-166.1811,0.0000
EC01322=-164.9600,0.0000
EC01323=-163.3682,0.0000
EC01324=-161.6026,0.0000
EC01325=-159.8845,0.0000
EC01326=-158.2829,0.0000
EC01327=-156.7174,0.0000
EC01328=-155.1153,0.0000
EC01329=-153.3978,0.0000
EC01330=-151.6323,0.0000
EC01331=-150.0400,0.0000
EC01332=-148.8185,0.0000
EC01333=-147.8519,0.0000
EC01334=-146.8911,0.0000
EC01335=-145.6851,0.0000
EC01336=-143.8992,0.0000
EC01337=-141.2433,0.0000
EC01338=-138.2710,0.0000
EC01339=-135.0000,0.0000
EC01340=-131.7290,0.0000
EC01341=-128.7567,0.0000
EC01342=-126.1008,0.0000
EC01343=-124.3149,0.0000
EC01344=-123.1089,0.0000
EC01345=-122.1481,0.0000
EC01346=-121.1815,0.0000
EC01347=-119.9600,0.0000
EC01348=-118.3677,0.0000
EC01349=-116.6022,0.0000
EC01350=-114.8847,0.0000
EC01351=-113.2826,0.0000
EC01352=-111.7171,0.0000
EC01353=-110.1155,0.0000
EC01354=-108.3974,0.0000
EC01355=-106.6318,0.0000
EC01356=-105.0400,0.0000
EC01357=-103.8189,0.0000
EC01358=-102.8520,0.0000
EC01359=-101.8912,0.0000
EC01360=-100.6850,0.0000
EC01361=-98.8988,0.0000
EC01362=-96.2435,0.0000
EC01363=-93.2709,0.0000
EC01364=-90.0000,0.0000
EC01365=-86.7291,0.0000
EC01366=-83.7565,0.0000
EC01367=-81.1012,0.0000
EC01368=-79.3150,0.0000
EC01369=-78.1088,0.0000
EC01370=-77.1480,0.0000
EC01371=-76.1811,0.0000
EC01372=-74.9600,0.0000
EC01373=-73.3682,0.0000
EC01374=-71.6026,0.0000
EC01375=-69.8845,0.0000
EC01376=-68.2829,0.0000
EC01377=-66.7174,0.0000
EC01378=-65.1153,0.0000
EC01379=-63.3978,0.0000
EC01380=-61.6323,0.0000
EC01381=-60.0400,0.0000
EC01382=-58.8185,0.0000
EC01383=-57.8519,0.0000
EC01384=-56.8911,0.0000
EC01385=-55.6851,0.0000
EC01386=-53.8992,0.0000
EC01387=-51.2433,0.0000
EC01388=-48.2710,0.0000
EC01389=-45.0000,0.0000
EC01390=-41.7290,0.0000
EC01391=-38.7567,0.0000
EC01392=-36.1008,0.0000
EC01393=-34.3149,0.0000
EC01394=-33.1089,0.0000
EC01395=-32.1481,0.0000
EC01396=-31.1815,0.0000
EC01397=-29.9600,0.0000
EC01398=-28.3677,0.0000
EC01399=-26.6022,0.0000
EC01400=-24.8847,0.0000
EC01401=-23.2826,0.0000
EC01402=-21.7171,0.0000
EC01403=-20.1155,0.0000
EC01404=-18.3974,0.0000
EC01405=-16.6318,0.0000
EC01406=-15.0400,0.0000
EC01407=-13.8189,0.0000
EC01408=-12.8520,0.0000
EC01409=-11.8912,0.0000
EC01410=-10.6850,0.0000
EC01411=-8.8988,0.0000
EC01412=-6.2435,0.0000
EC01413=-3.2709,0.0000
EC01414=0.0000,0.0000
EC01415=0.0000,0.0000
EC01416=3.2546,0.0000
EC01417=6.2211,0.0000
EC01418=8.8807,0.0000
EC01419=10.6541,0.0000
EC01420=11.8420,0.0000
EC01421=12.7823,0.0000
EC01422=13.7251,0.0000
EC01423=14.9190,0.0000
EC01424=16.5054,0.0000
EC01425=18.2889,0.0000
EC01426=20.0438,0.0000
EC01427=21.6927,0.0000
EC01428=23.3075,0.0000
EC01429=24.9564,0.0000
EC01430=26.7113,0.0000
EC01431=28.4943,0.0000
EC01432=30.0807,0.0000
EC01433=31.2747,0.0000
EC01434=32.2172,0.0000
EC01435=33.1579,0.0000
EC01436=34.3457,0.0000
EC01437=36.1194,0.0000
EC01438=38.7787,0.0000
EC01439=41.7455,0.0000
EC01440=45.0000,0.0000
EC01441=48.2545,0.0000
EC01442=51.2213,0.0000
EC01443=53.8806,0.0000
EC01444=55.6543,0.0000
EC01445=56.8421,0.0000
EC01446=57.7828,0.0000
EC01447=58.7253,0.0000
EC01448=59.9193,0.0000
EC01449=61.5057,0.0000
EC01450=63.2887,0.0000
EC01451=65.0436,0.0000
EC01452=66.6925,0.0000
EC01453=68.3073,0.0000
EC01454=69.9562,0.0000
EC01455=71.7111,0.0000
EC01456=73.4946,0.0000
EC01457=75.0810,0.0000
EC01458=76.2749,0.0000
EC01459=77.2177,0.0000
EC01460=78.1580,0.0000
EC01461=79.3459,0.0000
EC01462=81.1193,0.0000
EC01463=83.7789,0.0000
EC01464=86.7454,0.0000
EC01465=90.0000,0.0000
EC01466=93.2546,0.0000
EC01467=96.2211,0.0000
EC01468=98.8807,0.0000
EC01469=100.6541,0.0000
EC01470=101.8420,0.0000
EC01471=102.7823,0.0000
EC01472=103.7251,0.0000
EC01473=104.9190,0.0000
EC01474=106.5054,0.0000
EC01475=108.2889,0.0000
EC01476=110.0438,0.0000
EC01477=111.6927,0.0000
EC01478=113.3075,0.0000
EC01479=114.9564,0.0000
EC01480=116.7113,0.0000
EC01481=118.4943,0.0000
EC01482=120.0807,0.0000
EC01483=121.2747,0.0000
EC01484=122.2172,0.0000
EC01485=123.1579,0.0000
EC01486=124.3457,0.0000
EC01487=126.1194,0.0000
EC01488=128.7787,0.0000
EC01489=131.7455,0.0000
EC01490=135.0000,0.0000
EC01491=138.2545,0.0000
EC01492=141.2213,0.0000
EC01493=143.8806,0.0000
EC01494=145.6543,0.0000
EC01495=146.8421,0.0000
EC01496=147.7828,0.0000
EC01497=148.7253,0.0000
EC01498=149.9193,0.0000
EC01499=151.5057,0.0000
EC01500=153.2887,0.0000
EC01501=155.0436,0.0000
EC01502=156.6925,0.0000
EC01503=158.3073,0.0000
EC01504=159.9562,0.0000
EC01505=161.7111,0.0000
EC01506=163.4946,0.0000
EC01507=165.0810,0.0000
EC01508=166.2749,0.0000
EC01509=167.2177,0.0000
EC01510=168.1580,0.0000
EC01511=169.3459,0.0000
EC01512=171.1193,0.0000
EC01513=173.7789,0.0000
EC01514=176.7454,0.0000
EC01515=180.0000,0.0000
EC01516=180.0000,0.0000
EC01517=-176.7454,0.0000
EC01518=-173.7789,0.0000
EC01519=-171.1193,0.0000
EC01520=-169.3459,0.0000
EC01521=-168.1580,0.0000
EC01522=-167.2177,0.0000
EC01523=-166.2749,0.0000
EC01524=-165.0810,0.0000
EC01525=-163.4946,0.0000
EC01526=-161.7111,0.0000
EC01527=-159.9562,0.0000
EC01528=-158.3073,0.0000
EC01529=-156.6925,0.0000
EC01530=-155.0436,0.0000
EC01531=-153.2887,0.0000
EC01532=-151.5057,0.0000
EC01533=-149.9193,0.0000
EC01534=-148.7253,0.0000
EC01535=-147.7828,0.0000
EC01536=-146.8421,0.0000
EC01537=-145.6543,0.0000
EC01538=-143.8806,0.0000
EC01539=-141.2213,0.0000
EC01540=-138.2545,0.0000
EC01541=-135.0000,0.0000
EC01542=-131.7455,0.0000
EC01543=-128.7787,0.0000
EC01544=-126.1194,0.0000
EC01545=-124.3457,0.0000
EC01546=-123.1579,0.0000
EC01547=-122.2172,0.0000
EC01548=-121.2747,0.0000
EC01549=-120.0807,0.0000
EC01550=-118.4943,0.0000
EC01551=-116.7113,0.0000
EC01552=-114.9564,0.0000
EC01553=-113.3075,0.0000
EC01554=-111.6927,0.0000
EC01555=-110.0438,0.0000
EC01556=-108.2889,0.0000
EC01557=-106.5054,0.0000
EC01558=-104.9190,0.0000
EC01559=-103.7251,0.0000
EC01560=-102.7823,0.0000
EC01561=-101.8420,0.0000
EC01562=-100.6541,0.0000
EC01563=-98.8807,0.0000
EC01564=-96.2211,0.0000
EC01565=-93.2546,0.0000
EC01566=-90.0000,0.0000
EC01567=-86.7454,0.0000
EC01568=-83.7789,0.0000
EC01569=-81.1193,0.0000
EC01570=-79.3459,0.0000
EC01571=-78.1580,0.0000
EC01572=-77.2177,0.0000
EC01573=-76.2749,0.0000
EC01574=-75.0810,0.0000
EC01575=-73.4946,0.0000
EC01576=-71.7111,0.0000
EC01577=-69.9562,0.0000
EC01578=-68.3073,0.0000
EC01579=-66.6925,0.0000
EC01580=-65.0436,0.0000
EC01581=-63.2887,0.0000
EC01582=-61.5057,0.0000
EC01583=-59.9193,0.0000
EC01584=-58.7253,0.0000
EC01585=-57.7828,0.0000
EC01586=-56.8421,0.0000
EC01587=-55.6543,0.0000
EC01588=-53.8806,0.0000
EC01589=-51.2213,0.0000
EC01590=-48.2545,0.0000
EC01591=-45.0000,0.0000
EC01592=-41.7455,0.0000
EC01593=-38.7787,0.0000
EC01594=-36.1194,0.0000
EC01595=-34.3457,0.0000
EC01596=-33.1579,0.0000
EC01597=-32.2172,0.0000
EC01598=-31.2747,0.0000
EC01599=-30.0807,0.0000
EC01600=-28.4943,0.0000
EC01601=-26.7113,0.0000
EC01602=-24.9564,0.0000
EC01603=-23.3075,0.0000
EC01604=-21.6927,0.0000
EC01605=-20.0438,0.0000
EC01606=-18.2889,0.0000
EC01607=-16.5054,0.0000
EC01608=-14.9190,0.0000
EC01609=-13.7251,0.0000
EC01610=-12.7823,0.0000
EC01611=-11.8420,0.0000
EC01612=-10.6541,0.0000
EC01613=-8.8807,0.0000
EC01614=-6.2211,0.0000
EC01615=-3.2546,0.0000
EC01616=0.0000,0.0000
EC01617=0.0000,0.0000
EC01618=3.2359,0.0000
EC01619=6.1970,0.0000
EC01620=8.8601,0.0000
EC01621=10.6197,0.0000
EC01622=11.7864,0.0000
EC01623=12.7041,0.0000
EC01624=13.6200,0.0000
EC01625=14.7831,0.0000
EC01626=16.3632,0.0000
EC01627=18.1666,0.0000
EC01628=19.9634,0.0000
EC01629=21.6649,0.0000
EC01630=23.3352,0.0000
EC01631=25.0366,0.0000
EC01632=26.8332,0.0000
EC01633=28.6370,0.0000
EC01634=30.2167,0.0000
EC01635=31.3801,0.0000
EC01636=32.2959,0.0000
EC01637=33.2134,0.0000
EC01638=34.3801,0.0000
EC01639=36.1402,0.0000
EC01640=38.8032,0.0000
EC01641=41.7642,0.0000
EC01642=45.0000,0.0000
EC01643=48.2358,0.0000
EC01644=51.1968,0.0000
EC01645=53.8598,0.0000
EC01646=55.6199,0.0000
EC01647=56.7866,0.0000
EC01648=57.7041,0.0000
EC01649=58.6199,0.0000
EC01650=59.7833,0.0000
EC01651=61.3630,0.0000
EC01652=63.1668,0.0000
EC01653=64.9634,0.0000
EC01654=66.6648,0.0000
EC01655=68.3351,0.0000
EC01656=70.0366,0.0000
EC01657=71.8334,0.0000
EC01658=73.6368,0.0000
EC01659=75.2169,0.0000
EC01660=76.3800,0.0000
EC01661=77.2959,0.0000
EC01662=78.2136,0.0000
EC01663=79.3803,0.0000
EC01664=81.1399,0.0000
EC01665=83.8030,0.0000
EC01666=86.7641,0.0000
EC01667=90.0000,0.0000
EC01668=93.2359,0.0000
EC01669=96.1970,0.0000
EC01670=98.8601,0.0000
EC01671=100.6197,0.0000
EC01672=101.7864,0.0000
EC01673=102.7041,0.0000
EC01674=103.6200,0.0000
EC01675=104.7831,0.0000
EC01676=106.3632,0.0000
EC01677=108.1666,0.0000
EC01678=109.9634,0.0000
EC01679=111.6649,0.0000
EC01680=113.3352,0.0000
EC01681=115.0366,0.0000
EC01682=116.8332,0.0000
EC01683=118.6370,0.0000
EC01684=120.2167,0.0000
EC01685=121.3801,0.0000
EC01686=122.2959,0.0000
EC01687=123.2134,0.0000
EC01688=124.3801,0.0000
EC01689=126.1402,0.0000
EC01690=128.8032,0.0000
EC01691=131.7642,0.0000
EC01692=135.0000,0.0000
EC01693=138.2358,0.0000
EC01694=141.1968,0.0000
EC01695=143.8598,0.0000
EC01696=145.6199,0.0000
EC01697=146.7866,0.0000
EC01698=147.7041,0.0000
EC01699=148.6199,0.0000
EC01700=149.7833,0.0000
EC01701=151.3630,0.0000
EC01702=153.1668,0.0000
EC01703=154.9634,0.0000
EC01704=156.6648,0.0000
EC01705=158.3351,0.0000
EC01706=160.0366,0.0000
EC01707=161.8334,0.0000
EC01708=163.6368,0.0000
EC01709=165.2169,0.0000
EC01710=166.3800,0.0000
EC01711=167.2959,0.0000
EC01712=168.2136,0.0000
EC01713=169.3803,0.0000
EC01714=171.1399,0.0000
EC01715=173.8030,0.0000
EC01716=176.7641,0.0000
EC01717=180.0000,0.0000
EC01718=180.0000,0.0000
EC01719=-176.7641,0.0000
EC01720=-173.8030,0.0000
EC01721=-171.1399,0.0000
EC01722=-169.3803,0.0000
EC01723=-168.2136,0.0000
EC01724=-167.2959,0.0000
EC01725=-166.3800,0.0000
EC01726=-165.2169,0.0000
EC01727=-163.6368,0.0000
EC01728=-161.8334,0.0000
EC01729=-160.0366,0.0000
EC01730=-158.3351,0.0000
EC01731=-156.6648,0.0000
EC01732=-154.9634,0.0000
EC01733=-153.1668,0.0000
EC01734=-151.3630,0.0000
EC01735=-149.7833,0.0000
EC01736=-148.6199,0.0000
EC01737=-147.7041,0.0000
EC01738=-146.7866,0.0000
EC01739=-145.6199,0.0000
EC01740=-143.8598,0.0000
EC01741=-141.1968,0.0000
EC01742=-138.2358,0.0000
EC01743=-135.0000,0.0000
EC01744=-131.7642,0.0000
EC01745=-128.8032,0.0000
EC01746=-126.1402,0.0000
EC01747=-124.3801,0.0000
EC01748=-123.2134,0.0000
EC01749=-122.2959,0.0000
EC01750=-121.3801,0.0000
EC01751=-120.2167,0.0000
EC01752=-118.6370,0.0000
EC01753=-116.8332,0.0000
EC01754=-115.0366,0.0000
EC01755=-113.3352,0.0000
EC01756=-111.6649,0.0000
EC01757=-109.9634,0.0000
EC01758=-108.1666,0.0000
EC01759=-106.3632,0.0000
EC01760=-104.7831,0.0000
EC01761=-103.6200,0.0000
EC01762=-102.7041,0.0000
EC01763=-101.7864,0.0000
EC01764=-100.6197,0.0000
EC01765=-98.8601,0.0000
EC01766=-96.1970,0.0000
EC01767=-93.2359,0.0000
EC01768=-90.0000,0.0000
EC01769=-86.7641,0.0000
EC01770=-83.8030,0.0000
EC01771=-81.1399,0.0000
EC01772=-79.3803,0.0000
EC01773=-78.2136,0.0000
EC01774=-77.2959,0.0000
EC01775=-76.3800,0.0000
EC01776=-75.2169,0.0000
EC01777=-73.6368,0.0000
EC01778=-71.8334,0.0000
EC01779=-70.0366,0.0000
EC01780=-68.3351,0.0000
EC01781=-66.6648,0.0000
EC01782=-64.9634,0.0000
EC01783=-63.1668,0.0000
EC01784=-61.3630,0.0000
EC01785=-59.7833,0.0000
EC01786=-58.6199,0.0000
EC01787=-57.7041,0.0000
EC01788=-56.7866,0.0000
EC01789=-55.6199,0.0000
EC01790=-53.8598,0.0000
EC01791=-51.1968,0.0000
EC01792=-48.2358,0.0000
EC01793=-45.0000,0.0000
EC01794=-41.7642,0.0000
EC01795=-38.8032,0.0000
EC01796=-36.1402,0.0000
EC01797=-34.3801,0.0000
EC01798=-33.2134,0.0000
EC01799=-32.2959,0.0000
EC01800=-31.3801,0.0000
EC01801=-30.2167,0.0000
EC01802=-28.6370,0.0000
EC01803=-26.8332,0.0000
EC01804=-25.0366,0.0000
EC01805=-23.3352,0.0000
EC01806=-21.6649,0.0000
EC01807=-19.9634,0.0000
EC01808=-18.1666,0.0000
EC01809=-16.3632,0.0000
EC01810=-14.7831,0.0000
EC01811=-13.6200,0.0000
EC01812=-12.7041,0.0000
EC01813=-11.7864,0.0000
EC01814=-10.6197,0.0000
EC01815=-8.8601,0.0000
EC01816=-6.1970,0.0000
EC01817=-3.2359,0.0000
EC01818=0.0000,0.0000
EC01819=0.0000,0.0000
EC01820=3.2152,0.0000
EC01821=6.1699,0.0000
EC01822=8.8371,0.0000
EC01823=10.5819,0.0000
EC01824=11.7253,0.0000
EC01825=12.6169,0.0000
EC01826=13.5035,0.0000
EC01827=14.6333,0.0000
EC01828=16.2063,0.0000
EC01829=18.0324,0.0000
EC01830=19.8748,0.0000
EC01831=21.6343,0.0000
EC01832=23.3660,0.0000
EC01833=25.1253,0.0000
EC01834=26.9678,0.0000
EC01835=28.7935,0.0000
EC01836=30.3670,0.0000
EC01837=31.4965,0.0000
EC01838=32.3830,0.0000
EC01839=33.2751,0.0000
EC01840=34.4183,0.0000
EC01841=36.1625,0.0000
EC01842=38.8301,0.0000
EC01843=41.7846,0.0000
EC01844=45.0000,0.0000
EC01845=48.2154,0.0000
EC01846=51.1699,0.0000
EC01847=53.8375,0.0000
EC01848=55.5817,0.0000
EC01849=56.7249,0.0000
EC01850=57.6170,0.0000
EC01851=58.5035,0.0000
EC01852=59.6330,0.0000
EC01853=61.2065,0.0000
EC01854=63.0322,0.0000
EC01855=64.8747,0.0000
EC01856=66.6340,0.0000
EC01857=68.3657,0.0000
EC01858=70.1252,0.0000
EC01859=71.9676,0.0000
EC01860=73.7937,0.0000
EC01861=75.3667,0.0000
EC01862=76.4965,0.0000
EC01863=77.3831,0.0000
EC01864=78.2747,0.0000
EC01865=79.4181,0.0000
EC01866=81.1629,0.0000
EC01867=83.8301,0.0000
EC01868=86.7848,0.0000
EC01869=90.0000,0.0000
EC01870=93.2152,0.0000
EC01871=96.1699,0.0000
EC01872=98.8371,0.0000
EC01873=100.5819,0.0000
EC01874=101.7253,0.0000
EC01875=102.6169,0.0000
EC01876=103.5035,0.0000
EC01877=104.6333,0.0000
EC01878=106.2063,0.0000
EC01879=108.0324,0.0000
EC01880=109.8748,0.0000
EC01881=111.6343,0.0000
EC01882=113.3660,0.0000
EC01883=115.1253,0.0000
EC01884=116.9678,0.0000
EC01885=118.7935,0.0000
EC01886=120.3670,0.0000
EC01887=121.4965,0.0000
EC01888=122.3830,0.0000
EC01889=123.2751,0.0000
EC01890=124.4183,0.0000
EC01891=126.1625,0.0000
EC01892=128.8301,0.0000
EC01893=131.7846,0.0000
EC01894=135.0000,0.0000
EC01895=138.2154,0.0000
EC01896=141.1699,0.0000
EC01897=143.8375,0.0000
EC01898=145.5817,0.0000
EC01899=146.7249,0.0000
EC01900=147.6170,0.0000
EC01901=148.5035,0.0000
EC01902=149.6330,0.0000
EC01903=151.2065,0.0000
EC01904=153.0322,0.0000
EC01905=154.8747,0.0000
EC01906=156.6340,0.0000
EC01907=158.3657,0.0000
EC01908=160.1252,0.0000
EC01909=161.9676,0.0000
EC01910=163.7937,0.0000
EC01911=165.3667,0.0000
EC01912=166.4965,0.0000
EC01913=167.3831,0.0000
EC01914=168.2747,0.0000
EC01915=169.4181,0.0000
EC01916=171.1629,0.0000
EC01917=173.8301,0.0000
EC01918=176.7848,0.0000
EC01919=180.0000,0.0000
EC01920=180.0000,0.0000
EC01921=-176.7848,0.0000
EC01922=-173.8301,0.0000
EC01923=-171.1629,0.0000
EC01924=-169.4181,0.0000
EC01925=-168.2747,0.0000
EC01926=-167.3831,0.0000
EC01927=-166.4965,0.0000
EC01928=-165.3667,0.0000
EC01929=-163.7937,0.0000
EC01930=-161.9676,0.0000
EC01931=-160.1252,0.0000
EC01932=-158.3657,0.0000
EC01933=-156.6340,0.0000
EC01934=-154.8747,0.0000
EC01935=-153.0322,0.0000
EC01936=-151.2065,0.0000
EC01937=-149.6330,0.0000
EC01938=-148.5035,0.0000
EC01939=-147.6170,0.0000
EC01940=-146.7249,0.0000
EC01941=-145.5817,0.0000
EC01942=-143.8375,0.0000
EC01943=-141.1699,0.0000
EC01944=-138.2154,0.0000
EC01945=-135.0000,0.0000
EC01946=-131.7846,0.0000
EC01947=-128.8301,0.0000
EC01948=-126.1625,0.0000
EC01949=-124.4183,0.0000
EC01950=-123.2751,0.0000
EC01951=-122.3830,0.0000
EC01952=-121.4965,0.0000
EC01953=-120.3670,0.0000
EC01954=-118.7935,0.0000
EC01955=-116.9678,0.0000
EC01956=-115.1253,0.0000
EC01957=-113.3660,0.0000
EC01958=-111.6343,0.0000
EC01959=-109.8748,0.0000
EC01960=-108.0324,0.0000
EC01961=-106.2063,0.0000
EC01962=-104.6333,0.0000
EC01963=-103.5035,0.0000
EC01964=-102.6169,0.0000
EC01965=-101.7253,0.0000
EC01966=-100.5819,0.0000
EC01967=-98.8371,0.0000
EC01968=-96.1699,0.0000
EC01969=-93.2152,0.0000
EC01970=-90.0000,0.0000
EC01971=-86.7848,0.0000
EC01972=-83.8301,0.0000
EC01973=-81.1629,0.0000
EC01974=-79.4181,0.0000
EC01975=-78.2747,0.0000
EC01976=-77.3831,0.0000
EC01977=-76.4965,0.0000
EC01978=-75.3667,0.0000
EC01979=-73.7937,0.0000
EC01980=-71.9676,0.0000
EC01981=-70.1252,0.0000
EC01982=-68.3657,0.0000
EC01983=-66.6340,0.0000
EC01984=-64.8747,0.0000
EC01985=-63.0322,0.0000
EC01986=-61.2065,0.0000
EC01987=-59.6330,0.0000
EC01988=-58.5035,0.0000
EC01989=-57.6170,0.0000
EC01990=-56.7249,0.0000
EC01991=-55.5817,0.0000
EC01992=-53.8375,0.0000
EC01993=-51.1699,0.0000
EC01994=-48.2154,0.0000
EC01995=-45.0000,0.0000
EC01996=-41.7846,0.0000
EC01997=-38.8301,0.0000
EC01998=-36.1625,0.0000
EC01999=-34.4183,0.0000
//INST
///DATE 2021/02/10 13:51
///COMM
///ATTR SC,RW,RJ
////FRAME USER 2
///GROUP1 RB1
///GROUP2 ST1
NOP
SPEED V=20.0
SMOVL C00000 +MOVJ EC00000
ARCON
SMOVL C00001 +MOVJ EC00001
SPEED V=19.0
SMOVL C00002 +MOVJ EC00002
SPEED V=18.0
SMOVL C00003 +MOVJ EC00003
SPEED V=17.0
SMOVL C00004 +MOVJ EC00004
SPEED V=16.0
SMOVL C00005 +MOVJ EC00005
SPEED V=15.0
SMOVL C00006 +MOVJ EC00006
SPEED V=14.0
SMOVL C00007 +MOVJ EC00007
SPEED V=13.0
SMOVL C00008 +MOVJ EC00008
SPEED V=12.0
SMOVL C00009 +MOVJ EC00009
SPEED V=11.0
SMOVL C00010 +MOVJ EC00010
SPEED V=10.0
SMOVL C00011 +MOVJ EC00011
SMOVL C00012 +MOVJ EC00012
SMOVL C00013 +MOVJ EC00013
SMOVL C00014 +MOVJ EC00014
SMOVL C00015 +MOVJ EC00015
SMOVL C00016 +MOVJ EC00016
SMOVL C00017 +MOVJ EC00017
SMOVL C00018 +MOVJ EC00018
SMOVL C00019 +MOVJ EC00019
SMOVL C00020 +MOVJ EC00020
SMOVL C00021 +MOVJ EC00021
SMOVL C00022 +MOVJ EC00022
SMOVL C00023 +MOVJ EC00023
SMOVL C00024 +MOVJ EC00024
SMOVL C00025 +MOVJ EC00025
SMOVL C00026 +MOVJ EC00026
SMOVL C00027 +MOVJ EC00027
SMOVL C00028 +MOVJ EC00028
SMOVL C00029 +MOVJ EC00029
SMOVL C00030 +MOVJ EC00030
SMOVL C00031 +MOVJ EC00031
SMOVL C00032 +MOVJ EC00032
SMOVL C00033 +MOVJ EC00033
SMOVL C00034 +MOVJ EC00034
SMOVL C00035 +MOVJ EC00035
SMOVL C00036 +MOVJ EC00036
SMOVL C00037 +MOVJ EC00037
SMOVL C00038 +MOVJ EC00038
SMOVL C00039 +MOVJ EC00039
SMOVL C00040 +MOVJ EC00040
SMOVL C00041 +MOVJ EC00041
SMOVL C00042 +MOVJ EC00042
SMOVL C00043 +MOVJ EC00043
SMOVL C00044 +MOVJ EC00044
SMOVL C00045 +MOVJ EC00045
SMOVL C00046 +MOVJ EC00046
SMOVL C00047 +MOVJ EC00047
SMOVL C00048 +MOVJ EC00048
SMOVL C00049 +MOVJ EC00049
SMOVL C00050 +MOVJ EC00050
SMOVL C00051 +MOVJ EC00051
SMOVL C00052 +MOVJ EC00052
SMOVL C00053 +MOVJ EC00053
SMOVL C00054 +MOVJ EC00054
SMOVL C00055 +MOVJ EC00055
SMOVL C00056 +MOVJ EC00056
SMOVL C00057 +MOVJ EC00057
SMOVL C00058 +MOVJ EC00058
SMOVL C00059 +MOVJ EC00059
SMOVL C00060 +MOVJ EC00060
SMOVL C00061 +MOVJ EC00061
SMOVL C00062 +MOVJ EC00062
SMOVL C00063 +MOVJ EC00063
SMOVL C00064 +MOVJ EC00064
SMOVL C00065 +MOVJ EC00065
SMOVL C00066 +MOVJ EC00066
SMOVL C00067 +MOVJ EC00067
SMOVL C00068 +MOVJ EC00068
SMOVL C00069 +MOVJ EC00069
SMOVL C00070 +MOVJ EC00070
SMOVL C00071 +MOVJ EC00071
SMOVL C00072 +MOVJ EC00072
SMOVL C00073 +MOVJ EC00073
SMOVL C00074 +MOVJ EC00074
SMOVL C00075 +MOVJ EC00075
SMOVL C00076 +MOVJ EC00076
SMOVL C00077 +MOVJ EC00077
SMOVL C00078 +MOVJ EC00078
SMOVL C00079 +MOVJ EC00079
SMOVL C00080 +MOVJ EC00080
SMOVL C00081 +MOVJ EC00081
SMOVL C00082 +MOVJ EC00082
SMOVL C00083 +MOVJ EC00083
SMOVL C00084 +MOVJ EC00084
SMOVL C00085 +MOVJ EC00085
SMOVL C00086 +MOVJ EC00086
SMOVL C00087 +MOVJ EC00087
SMOVL C00088 +MOVJ EC00088
SMOVL C00089 +MOVJ EC00089
SMOVL C00090 +MOVJ EC00090
SMOVL C00091 +MOVJ EC00091
SMOVL C00092 +MOVJ EC00092
SMOVL C00093 +MOVJ EC00093
SMOVL C00094 +MOVJ EC00094
SMOVL C00095 +MOVJ EC00095
SMOVL C00096 +MOVJ EC00096
SMOVL C00097 +MOVJ EC00097
SMOVL C00098 +MOVJ EC00098
SMOVL C00099 +MOVJ EC00099
SMOVL C00100 +MOVJ EC00100
SMOVL C00101 +MOVJ EC00101
SMOVL C00102 +MOVJ EC00102
SMOVL C00103 +MOVJ EC00103
SMOVL C00104 +MOVJ EC00104
SMOVL C00105 +MOVJ EC00105
SMOVL C00106 +MOVJ EC00106
SMOVL C00107 +MOVJ EC00107
SMOVL C00108 +MOVJ EC00108
SMOVL C00109 +MOVJ EC00109
SMOVL C00110 +MOVJ EC00110
SMOVL C00111 +MOVJ EC00111
SMOVL C00112 +MOVJ EC00112
SMOVL C00113 +MOVJ EC00113
SMOVL C00114 +MOVJ EC00114
SMOVL C00115 +MOVJ EC00115
SMOVL C00116 +MOVJ EC00116
SMOVL C00117 +MOVJ EC00117
SMOVL C00118 +MOVJ EC00118
SMOVL C00119 +MOVJ EC00119
SMOVL C00120 +MOVJ EC00120
SMOVL C00121 +MOVJ EC00121
SMOVL C00122 +MOVJ EC00122
SMOVL C00123 +MOVJ EC00123
SMOVL C00124 +MOVJ EC00124
SMOVL C00125 +MOVJ EC00125
SMOVL C00126 +MOVJ EC00126
SMOVL C00127 +MOVJ EC00127
SMOVL C00128 +MOVJ EC00128
SMOVL C00129 +MOVJ EC00129
SMOVL C00130 +MOVJ EC00130
SMOVL C00131 +MOVJ EC00131
SMOVL C00132 +MOVJ EC00132
SMOVL C00133 +MOVJ EC00133
SMOVL C00134 +MOVJ EC00134
SMOVL C00135 +MOVJ EC00135
SMOVL C00136 +MOVJ EC00136
SMOVL C00137 +MOVJ EC00137
SMOVL C00138 +MOVJ EC00138
SMOVL C00139 +MOVJ EC00139
SMOVL C00140 +MOVJ EC00140
SMOVL C00141 +MOVJ EC00141
SMOVL C00142 +MOVJ EC00142
SMOVL C00143 +MOVJ EC00143
SMOVL C00144 +MOVJ EC00144
SMOVL C00145 +MOVJ EC00145
SMOVL C00146 +MOVJ EC00146
SMOVL C00147 +MOVJ EC00147
SMOVL C00148 +MOVJ EC00148
SMOVL C00149 +MOVJ EC00149
SMOVL C00150 +MOVJ EC00150
SMOVL C00151 +MOVJ EC00151
SMOVL C00152 +MOVJ EC00152
SMOVL C00153 +MOVJ EC00153
SMOVL C00154 +MOVJ EC00154
SMOVL C00155 +MOVJ EC00155
SMOVL C00156 +MOVJ EC00156
SMOVL C00157 +MOVJ EC00157
SMOVL C00158 +MOVJ EC00158
SMOVL C00159 +MOVJ EC00159
SMOVL C00160 +MOVJ EC00160
SMOVL C00161 +MOVJ EC00161
SMOVL C00162 +MOVJ EC00162
SMOVL C00163 +MOVJ EC00163
SMOVL C00164 +MOVJ EC00164
SMOVL C00165 +MOVJ EC00165
SMOVL C00166 +MOVJ EC00166
SMOVL C00167 +MOVJ EC00167
SMOVL C00168 +MOVJ EC00168
SMOVL C00169 +MOVJ EC00169
SMOVL C00170 +MOVJ EC00170
SMOVL C00171 +MOVJ EC00171
SMOVL C00172 +MOVJ EC00172
SMOVL C00173 +MOVJ EC00173
SMOVL C00174 +MOVJ EC00174
SMOVL C00175 +MOVJ EC00175
SMOVL C00176 +MOVJ EC00176
SMOVL C00177 +MOVJ EC00177
SMOVL C00178 +MOVJ EC00178
SMOVL C00179 +MOVJ EC00179
SMOVL C00180 +MOVJ EC00180
SMOVL C00181 +MOVJ EC00181
SMOVL C00182 +MOVJ EC00182
SMOVL C00183 +MOVJ EC00183
SMOVL C00184 +MOVJ EC00184
SMOVL C00185 +MOVJ EC00185
SMOVL C00186 +MOVJ EC00186
SMOVL C00187 +MOVJ EC00187
SMOVL C00188 +MOVJ EC00188
SMOVL C00189 +MOVJ EC00189
SMOVL C00190 +MOVJ EC00190
SMOVL C00191 +MOVJ EC00191
SMOVL C00192 +MOVJ EC00192
SMOVL C00193 +MOVJ EC00193
SMOVL C00194 +MOVJ EC00194
SMOVL C00195 +MOVJ EC00195
SMOVL C00196 +MOVJ EC00196
SMOVL C00197 +MOVJ EC00197
SMOVL C00198 +MOVJ EC00198
SMOVL C00199 +MOVJ EC00199
SMOVL C00200 +MOVJ EC00200
SMOVL C00201 +MOVJ EC00201
SMOVL C00202 +MOVJ EC00202
SMOVL C00203 +MOVJ EC00203
SMOVL C00204 +MOVJ EC00204
SMOVL C00205 +MOVJ EC00205
SMOVL C00206 +MOVJ EC00206
SMOVL C00207 +MOVJ EC00207
SMOVL C00208 +MOVJ EC00208
SMOVL C00209 +MOVJ EC00209
SMOVL C00210 +MOVJ EC00210
SMOVL C00211 +MOVJ EC00211
SMOVL C00212 +MOVJ EC00212
SMOVL C00213 +MOVJ EC00213
SMOVL C00214 +MOVJ EC00214
SMOVL C00215 +MOVJ EC00215
SMOVL C00216 +MOVJ EC00216
SMOVL C00217 +MOVJ EC00217
SMOVL C00218 +MOVJ EC00218
SMOVL C00219 +MOVJ EC00219
SMOVL C00220 +MOVJ EC00220
SMOVL C00221 +MOVJ EC00221
SMOVL C00222 +MOVJ EC00222
SMOVL C00223 +MOVJ EC00223
SMOVL C00224 +MOVJ EC00224
SMOVL C00225 +MOVJ EC00225
SMOVL C00226 +MOVJ EC00226
SMOVL C00227 +MOVJ EC00227
SMOVL C00228 +MOVJ EC00228
SMOVL C00229 +MOVJ EC00229
SMOVL C00230 +MOVJ EC00230
SMOVL C00231 +MOVJ EC00231
SMOVL C00232 +MOVJ EC00232
SMOVL C00233 +MOVJ EC00233
SMOVL C00234 +MOVJ EC00234
SMOVL C00235 +MOVJ EC00235
SMOVL C00236 +MOVJ EC00236
SMOVL C00237 +MOVJ EC00237
SMOVL C00238 +MOVJ EC00238
SMOVL C00239 +MOVJ EC00239
SMOVL C00240 +MOVJ EC00240
SMOVL C00241 +MOVJ EC00241
SMOVL C00242 +MOVJ EC00242
SMOVL C00243 +MOVJ EC00243
SMOVL C00244 +MOVJ EC00244
SMOVL C00245 +MOVJ EC00245
SMOVL C00246 +MOVJ EC00246
SMOVL C00247 +MOVJ EC00247
SMOVL C00248 +MOVJ EC00248
SMOVL C00249 +MOVJ EC00249
SMOVL C00250 +MOVJ EC00250
SMOVL C00251 +MOVJ EC00251
SMOVL C00252 +MOVJ EC00252
SMOVL C00253 +MOVJ EC00253
SMOVL C00254 +MOVJ EC00254
SMOVL C00255 +MOVJ EC00255
SMOVL C00256 +MOVJ EC00256
SMOVL C00257 +MOVJ EC00257
SMOVL C00258 +MOVJ EC00258
SMOVL C00259 +MOVJ EC00259
SMOVL C00260 +MOVJ EC00260
SMOVL C00261 +MOVJ EC00261
SMOVL C00262 +MOVJ EC00262
SMOVL C00263 +MOVJ EC00263
SMOVL C00264 +MOVJ EC00264
SMOVL C00265 +MOVJ EC00265
SMOVL C00266 +MOVJ EC00266
SMOVL C00267 +MOVJ EC00267
SMOVL C00268 +MOVJ EC00268
SMOVL C00269 +MOVJ EC00269
SMOVL C00270 +MOVJ EC00270
SMOVL C00271 +MOVJ EC00271
SMOVL C00272 +MOVJ EC00272
SMOVL C00273 +MOVJ EC00273
SMOVL C00274 +MOVJ EC00274
SMOVL C00275 +MOVJ EC00275
SMOVL C00276 +MOVJ EC00276
SMOVL C00277 +MOVJ EC00277
SMOVL C00278 +MOVJ EC00278
SMOVL C00279 +MOVJ EC00279
SMOVL C00280 +MOVJ EC00280
SMOVL C00281 +MOVJ EC00281
SMOVL C00282 +MOVJ EC00282
SMOVL C00283 +MOVJ EC00283
SMOVL C00284 +MOVJ EC00284
SMOVL C00285 +MOVJ EC00285
SMOVL C00286 +MOVJ EC00286
SMOVL C00287 +MOVJ EC00287
SMOVL C00288 +MOVJ EC00288
SMOVL C00289 +MOVJ EC00289
SMOVL C00290 +MOVJ EC00290
SMOVL C00291 +MOVJ EC00291
SMOVL C00292 +MOVJ EC00292
SMOVL C00293 +MOVJ EC00293
SMOVL C00294 +MOVJ EC00294
SMOVL C00295 +MOVJ EC00295
SMOVL C00296 +MOVJ EC00296
SMOVL C00297 +MOVJ EC00297
SMOVL C00298 +MOVJ EC00298
SMOVL C00299 +MOVJ EC00299
SMOVL C00300 +MOVJ EC00300
SMOVL C00301 +MOVJ EC00301
SMOVL C00302 +MOVJ EC00302
SMOVL C00303 +MOVJ EC00303
SMOVL C00304 +MOVJ EC00304
SMOVL C00305 +MOVJ EC00305
SMOVL C00306 +MOVJ EC00306
SMOVL C00307 +MOVJ EC00307
SMOVL C00308 +MOVJ EC00308
SMOVL C00309 +MOVJ EC00309
SMOVL C00310 +MOVJ EC00310
SMOVL C00311 +MOVJ EC00311
SMOVL C00312 +MOVJ EC00312
SMOVL C00313 +MOVJ EC00313
SMOVL C00314 +MOVJ EC00314
SMOVL C00315 +MOVJ EC00315
SMOVL C00316 +MOVJ EC00316
SMOVL C00317 +MOVJ EC00317
SMOVL C00318 +MOVJ EC00318
SMOVL C00319 +MOVJ EC00319
SMOVL C00320 +MOVJ EC00320
SMOVL C00321 +MOVJ EC00321
SMOVL C00322 +MOVJ EC00322
SMOVL C00323 +MOVJ EC00323
SMOVL C00324 +MOVJ EC00324
SMOVL C00325 +MOVJ EC00325
SMOVL C00326 +MOVJ EC00326
SMOVL C00327 +MOVJ EC00327
SMOVL C00328 +MOVJ EC00328
SMOVL C00329 +MOVJ EC00329
SMOVL C00330 +MOVJ EC00330
SMOVL C00331 +MOVJ EC00331
SMOVL C00332 +MOVJ EC00332
SMOVL C00333 +MOVJ EC00333
SMOVL C00334 +MOVJ EC00334
SMOVL C00335 +MOVJ EC00335
SMOVL C00336 +MOVJ EC00336
SMOVL C00337 +MOVJ EC00337
SMOVL C00338 +MOVJ EC00338
SMOVL C00339 +MOVJ EC00339
SMOVL C00340 +MOVJ EC00340
SMOVL C00341 +MOVJ EC00341
SMOVL C00342 +MOVJ EC00342
SMOVL C00343 +MOVJ EC00343
SMOVL C00344 +MOVJ EC00344
SMOVL C00345 +MOVJ EC00345
SMOVL C00346 +MOVJ EC00346
SMOVL C00347 +MOVJ EC00347
SMOVL C00348 +MOVJ EC00348
SMOVL C00349 +MOVJ EC00349
SMOVL C00350 +MOVJ EC00350
SMOVL C00351 +MOVJ EC00351
SMOVL C00352 +MOVJ EC00352
SMOVL C00353 +MOVJ EC00353
SMOVL C00354 +MOVJ EC00354
SMOVL C00355 +MOVJ EC00355
SMOVL C00356 +MOVJ EC00356
SMOVL C00357 +MOVJ EC00357
SMOVL C00358 +MOVJ EC00358
SMOVL C00359 +MOVJ EC00359
SMOVL C00360 +MOVJ EC00360
SMOVL C00361 +MOVJ EC00361
SMOVL C00362 +MOVJ EC00362
SMOVL C00363 +MOVJ EC00363
SMOVL C00364 +MOVJ EC00364
SMOVL C00365 +MOVJ EC00365
SMOVL C00366 +MOVJ EC00366
SMOVL C00367 +MOVJ EC00367
SMOVL C00368 +MOVJ EC00368
SMOVL C00369 +MOVJ EC00369
SMOVL C00370 +MOVJ EC00370
SMOVL C00371 +MOVJ EC00371
SMOVL C00372 +MOVJ EC00372
SMOVL C00373 +MOVJ EC00373
SMOVL C00374 +MOVJ EC00374
SMOVL C00375 +MOVJ EC00375
SMOVL C00376 +MOVJ EC00376
SMOVL C00377 +MOVJ EC00377
SMOVL C00378 +MOVJ EC00378
SMOVL C00379 +MOVJ EC00379
SMOVL C00380 +MOVJ EC00380
SMOVL C00381 +MOVJ EC00381
SMOVL C00382 +MOVJ EC00382
SMOVL C00383 +MOVJ EC00383
SMOVL C00384 +MOVJ EC00384
SMOVL C00385 +MOVJ EC00385
SMOVL C00386 +MOVJ EC00386
SMOVL C00387 +MOVJ EC00387
SMOVL C00388 +MOVJ EC00388
SMOVL C00389 +MOVJ EC00389
SMOVL C00390 +MOVJ EC00390
SMOVL C00391 +MOVJ EC00391
SMOVL C00392 +MOVJ EC00392
SMOVL C00393 +MOVJ EC00393
SMOVL C00394 +MOVJ EC00394
SMOVL C00395 +MOVJ EC00395
SMOVL C00396 +MOVJ EC00396
SMOVL C00397 +MOVJ EC00397
SMOVL C00398 +MOVJ EC00398
SMOVL C00399 +MOVJ EC00399
SMOVL C00400 +MOVJ EC00400
SMOVL C00401 +MOVJ EC00401
SMOVL C00402 +MOVJ EC00402
SMOVL C00403 +MOVJ EC00403
SMOVL C00404 +MOVJ EC00404
SMOVL C00405 +MOVJ EC00405
SMOVL C00406 +MOVJ EC00406
SMOVL C00407 +MOVJ EC00407
SMOVL C00408 +MOVJ EC00408
SMOVL C00409 +MOVJ EC00409
SMOVL C00410 +MOVJ EC00410
SMOVL C00411 +MOVJ EC00411
SMOVL C00412 +MOVJ EC00412
SMOVL C00413 +MOVJ EC00413
SMOVL C00414 +MOVJ EC00414
SMOVL C00415 +MOVJ EC00415
SMOVL C00416 +MOVJ EC00416
SMOVL C00417 +MOVJ EC00417
SMOVL C00418 +MOVJ EC00418
SMOVL C00419 +MOVJ EC00419
SMOVL C00420 +MOVJ EC00420
SMOVL C00421 +MOVJ EC00421
SMOVL C00422 +MOVJ EC00422
SMOVL C00423 +MOVJ EC00423
SMOVL C00424 +MOVJ EC00424
SMOVL C00425 +MOVJ EC00425
SMOVL C00426 +MOVJ EC00426
SMOVL C00427 +MOVJ EC00427
SMOVL C00428 +MOVJ EC00428
SMOVL C00429 +MOVJ EC00429
SMOVL C00430 +MOVJ EC00430
SMOVL C00431 +MOVJ EC00431
SMOVL C00432 +MOVJ EC00432
SMOVL C00433 +MOVJ EC00433
SMOVL C00434 +MOVJ EC00434
SMOVL C00435 +MOVJ EC00435
SMOVL C00436 +MOVJ EC00436
SMOVL C00437 +MOVJ EC00437
SMOVL C00438 +MOVJ EC00438
SMOVL C00439 +MOVJ EC00439
SMOVL C00440 +MOVJ EC00440
SMOVL C00441 +MOVJ EC00441
SMOVL C00442 +MOVJ EC00442
SMOVL C00443 +MOVJ EC00443
SMOVL C00444 +MOVJ EC00444
SMOVL C00445 +MOVJ EC00445
SMOVL C00446 +MOVJ EC00446
SMOVL C00447 +MOVJ EC00447
SMOVL C00448 +MOVJ EC00448
SMOVL C00449 +MOVJ EC00449
SMOVL C00450 +MOVJ EC00450
SMOVL C00451 +MOVJ EC00451
SMOVL C00452 +MOVJ EC00452
SMOVL C00453 +MOVJ EC00453
SMOVL C00454 +MOVJ EC00454
SMOVL C00455 +MOVJ EC00455
SMOVL C00456 +MOVJ EC00456
SMOVL C00457 +MOVJ EC00457
SMOVL C00458 +MOVJ EC00458
SMOVL C00459 +MOVJ EC00459
SMOVL C00460 +MOVJ EC00460
SMOVL C00461 +MOVJ EC00461
SMOVL C00462 +MOVJ EC00462
SMOVL C00463 +MOVJ EC00463
SMOVL C00464 +MOVJ EC00464
SMOVL C00465 +MOVJ EC00465
SMOVL C00466 +MOVJ EC00466
SMOVL C00467 +MOVJ EC00467
SMOVL C00468 +MOVJ EC00468
SMOVL C00469 +MOVJ EC00469
SMOVL C00470 +MOVJ EC00470
SMOVL C00471 +MOVJ EC00471
SMOVL C00472 +MOVJ EC00472
SMOVL C00473 +MOVJ EC00473
SMOVL C00474 +MOVJ EC00474
SMOVL C00475 +MOVJ EC00475
SMOVL C00476 +MOVJ EC00476
SMOVL C00477 +MOVJ EC00477
SMOVL C00478 +MOVJ EC00478
SMOVL C00479 +MOVJ EC00479
SMOVL C00480 +MOVJ EC00480
SMOVL C00481 +MOVJ EC00481
SMOVL C00482 +MOVJ EC00482
SMOVL C00483 +MOVJ EC00483
SMOVL C00484 +MOVJ EC00484
SMOVL C00485 +MOVJ EC00485
SMOVL C00486 +MOVJ EC00486
SMOVL C00487 +MOVJ EC00487
SMOVL C00488 +MOVJ EC00488
SMOVL C00489 +MOVJ EC00489
SMOVL C00490 +MOVJ EC00490
SMOVL C00491 +MOVJ EC00491
SMOVL C00492 +MOVJ EC00492
SMOVL C00493 +MOVJ EC00493
SMOVL C00494 +MOVJ EC00494
SMOVL C00495 +MOVJ EC00495
SMOVL C00496 +MOVJ EC00496
SMOVL C00497 +MOVJ EC00497
SMOVL C00498 +MOVJ EC00498
SMOVL C00499 +MOVJ EC00499
SMOVL C00500 +MOVJ EC00500
SMOVL C00501 +MOVJ EC00501
SMOVL C00502 +MOVJ EC00502
SMOVL C00503 +MOVJ EC00503
SMOVL C00504 +MOVJ EC00504
SMOVL C00505 +MOVJ EC00505
SMOVL C00506 +MOVJ EC00506
SMOVL C00507 +MOVJ EC00507
SMOVL C00508 +MOVJ EC00508
SMOVL C00509 +MOVJ EC00509
SMOVL C00510 +MOVJ EC00510
SMOVL C00511 +MOVJ EC00511
SMOVL C00512 +MOVJ EC00512
SMOVL C00513 +MOVJ EC00513
SMOVL C00514 +MOVJ EC00514
SMOVL C00515 +MOVJ EC00515
SMOVL C00516 +MOVJ EC00516
SMOVL C00517 +MOVJ EC00517
SMOVL C00518 +MOVJ EC00518
SMOVL C00519 +MOVJ EC00519
SMOVL C00520 +MOVJ EC00520
SMOVL C00521 +MOVJ EC00521
SMOVL C00522 +MOVJ EC00522
SMOVL C00523 +MOVJ EC00523
SMOVL C00524 +MOVJ EC00524
SMOVL C00525 +MOVJ EC00525
SMOVL C00526 +MOVJ EC00526
SMOVL C00527 +MOVJ EC00527
SMOVL C00528 +MOVJ EC00528
SMOVL C00529 +MOVJ EC00529
SMOVL C00530 +MOVJ EC00530
SMOVL C00531 +MOVJ EC00531
SMOVL C00532 +MOVJ EC00532
SMOVL C00533 +MOVJ EC00533
SMOVL C00534 +MOVJ EC00534
SMOVL C00535 +MOVJ EC00535
SMOVL C00536 +MOVJ EC00536
SMOVL C00537 +MOVJ EC00537
SMOVL C00538 +MOVJ EC00538
SMOVL C00539 +MOVJ EC00539
SMOVL C00540 +MOVJ EC00540
SMOVL C00541 +MOVJ EC00541
SMOVL C00542 +MOVJ EC00542
SMOVL C00543 +MOVJ EC00543
SMOVL C00544 +MOVJ EC00544
SMOVL C00545 +MOVJ EC00545
SMOVL C00546 +MOVJ EC00546
SMOVL C00547 +MOVJ EC00547
SMOVL C00548 +MOVJ EC00548
SMOVL C00549 +MOVJ EC00549
SMOVL C00550 +MOVJ EC00550
SMOVL C00551 +MOVJ EC00551
SMOVL C00552 +MOVJ EC00552
SMOVL C00553 +MOVJ EC00553
SMOVL C00554 +MOVJ EC00554
SMOVL C00555 +MOVJ EC00555
SMOVL C00556 +MOVJ EC00556
SMOVL C00557 +MOVJ EC00557
SMOVL C00558 +MOVJ EC00558
SMOVL C00559 +MOVJ EC00559
SMOVL C00560 +MOVJ EC00560
SMOVL C00561 +MOVJ EC00561
SMOVL C00562 +MOVJ EC00562
SMOVL C00563 +MOVJ EC00563
SMOVL C00564 +MOVJ EC00564
SMOVL C00565 +MOVJ EC00565
SMOVL C00566 +MOVJ EC00566
SMOVL C00567 +MOVJ EC00567
SMOVL C00568 +MOVJ EC00568
SMOVL C00569 +MOVJ EC00569
SMOVL C00570 +MOVJ EC00570
SMOVL C00571 +MOVJ EC00571
SMOVL C00572 +MOVJ EC00572
SMOVL C00573 +MOVJ EC00573
SMOVL C00574 +MOVJ EC00574
SMOVL C00575 +MOVJ EC00575
SMOVL C00576 +MOVJ EC00576
SMOVL C00577 +MOVJ EC00577
SMOVL C00578 +MOVJ EC00578
SMOVL C00579 +MOVJ EC00579
SMOVL C00580 +MOVJ EC00580
SMOVL C00581 +MOVJ EC00581
SMOVL C00582 +MOVJ EC00582
SMOVL C00583 +MOVJ EC00583
SMOVL C00584 +MOVJ EC00584
SMOVL C00585 +MOVJ EC00585
SMOVL C00586 +MOVJ EC00586
SMOVL C00587 +MOVJ EC00587
SMOVL C00588 +MOVJ EC00588
SMOVL C00589 +MOVJ EC00589
SMOVL C00590 +MOVJ EC00590
SMOVL C00591 +MOVJ EC00591
SMOVL C00592 +MOVJ EC00592
SMOVL C00593 +MOVJ EC00593
SMOVL C00594 +MOVJ EC00594
SMOVL C00595 +MOVJ EC00595
SMOVL C00596 +MOVJ EC00596
SMOVL C00597 +MOVJ EC00597
SMOVL C00598 +MOVJ EC00598
SMOVL C00599 +MOVJ EC00599
SMOVL C00600 +MOVJ EC00600
SMOVL C00601 +MOVJ EC00601
SMOVL C00602 +MOVJ EC00602
SMOVL C00603 +MOVJ EC00603
SMOVL C00604 +MOVJ EC00604
SMOVL C00605 +MOVJ EC00605
SMOVL C00606 +MOVJ EC00606
SMOVL C00607 +MOVJ EC00607
SMOVL C00608 +MOVJ EC00608
SMOVL C00609 +MOVJ EC00609
SMOVL C00610 +MOVJ EC00610
SMOVL C00611 +MOVJ EC00611
SMOVL C00612 +MOVJ EC00612
SMOVL C00613 +MOVJ EC00613
SMOVL C00614 +MOVJ EC00614
SMOVL C00615 +MOVJ EC00615
SMOVL C00616 +MOVJ EC00616
SMOVL C00617 +MOVJ EC00617
SMOVL C00618 +MOVJ EC00618
SMOVL C00619 +MOVJ EC00619
SMOVL C00620 +MOVJ EC00620
SMOVL C00621 +MOVJ EC00621
SMOVL C00622 +MOVJ EC00622
SMOVL C00623 +MOVJ EC00623
SMOVL C00624 +MOVJ EC00624
SMOVL C00625 +MOVJ EC00625
SMOVL C00626 +MOVJ EC00626
SMOVL C00627 +MOVJ EC00627
SMOVL C00628 +MOVJ EC00628
SMOVL C00629 +MOVJ EC00629
SMOVL C00630 +MOVJ EC00630
SMOVL C00631 +MOVJ EC00631
SMOVL C00632 +MOVJ EC00632
SMOVL C00633 +MOVJ EC00633
SMOVL C00634 +MOVJ EC00634
SMOVL C00635 +MOVJ EC00635
SMOVL C00636 +MOVJ EC00636
SMOVL C00637 +MOVJ EC00637
SMOVL C00638 +MOVJ EC00638
SMOVL C00639 +MOVJ EC00639
SMOVL C00640 +MOVJ EC00640
SMOVL C00641 +MOVJ EC00641
SMOVL C00642 +MOVJ EC00642
SMOVL C00643 +MOVJ EC00643
SMOVL C00644 +MOVJ EC00644
SMOVL C00645 +MOVJ EC00645
SMOVL C00646 +MOVJ EC00646
SMOVL C00647 +MOVJ EC00647
SMOVL C00648 +MOVJ EC00648
SMOVL C00649 +MOVJ EC00649
SMOVL C00650 +MOVJ EC00650
SMOVL C00651 +MOVJ EC00651
SMOVL C00652 +MOVJ EC00652
SMOVL C00653 +MOVJ EC00653
SMOVL C00654 +MOVJ EC00654
SMOVL C00655 +MOVJ EC00655
SMOVL C00656 +MOVJ EC00656
SMOVL C00657 +MOVJ EC00657
SMOVL C00658 +MOVJ EC00658
SMOVL C00659 +MOVJ EC00659
SMOVL C00660 +MOVJ EC00660
SMOVL C00661 +MOVJ EC00661
SMOVL C00662 +MOVJ EC00662
SMOVL C00663 +MOVJ EC00663
SMOVL C00664 +MOVJ EC00664
SMOVL C00665 +MOVJ EC00665
SMOVL C00666 +MOVJ EC00666
SMOVL C00667 +MOVJ EC00667
SMOVL C00668 +MOVJ EC00668
SMOVL C00669 +MOVJ EC00669
SMOVL C00670 +MOVJ EC00670
SMOVL C00671 +MOVJ EC00671
SMOVL C00672 +MOVJ EC00672
SMOVL C00673 +MOVJ EC00673
SMOVL C00674 +MOVJ EC00674
SMOVL C00675 +MOVJ EC00675
SMOVL C00676 +MOVJ EC00676
SMOVL C00677 +MOVJ EC00677
SMOVL C00678 +MOVJ EC00678
SMOVL C00679 +MOVJ EC00679
SMOVL C00680 +MOVJ EC00680
SMOVL C00681 +MOVJ EC00681
SMOVL C00682 +MOVJ EC00682
SMOVL C00683 +MOVJ EC00683
SMOVL C00684 +MOVJ EC00684
SMOVL C00685 +MOVJ EC00685
SMOVL C00686 +MOVJ EC00686
SMOVL C00687 +MOVJ EC00687
SMOVL C00688 +MOVJ EC00688
SMOVL C00689 +MOVJ EC00689
SMOVL C00690 +MOVJ EC00690
SMOVL C00691 +MOVJ EC00691
SMOVL C00692 +MOVJ EC00692
SMOVL C00693 +MOVJ EC00693
SMOVL C00694 +MOVJ EC00694
SMOVL C00695 +MOVJ EC00695
SMOVL C00696 +MOVJ EC00696
SMOVL C00697 +MOVJ EC00697
SMOVL C00698 +MOVJ EC00698
SMOVL C00699 +MOVJ EC00699
SMOVL C00700 +MOVJ EC00700
SMOVL C00701 +MOVJ EC00701
SMOVL C00702 +MOVJ EC00702
SMOVL C00703 +MOVJ EC00703
SMOVL C00704 +MOVJ EC00704
SMOVL C00705 +MOVJ EC00705
SMOVL C00706 +MOVJ EC00706
SMOVL C00707 +MOVJ EC00707
SMOVL C00708 +MOVJ EC00708
SMOVL C00709 +MOVJ EC00709
SMOVL C00710 +MOVJ EC00710
SMOVL C00711 +MOVJ EC00711
SMOVL C00712 +MOVJ EC00712
SMOVL C00713 +MOVJ EC00713
SMOVL C00714 +MOVJ EC00714
SMOVL C00715 +MOVJ EC00715
SMOVL C00716 +MOVJ EC00716
SMOVL C00717 +MOVJ EC00717
SMOVL C00718 +MOVJ EC00718
SMOVL C00719 +MOVJ EC00719
SMOVL C00720 +MOVJ EC00720
SMOVL C00721 +MOVJ EC00721
SMOVL C00722 +MOVJ EC00722
SMOVL C00723 +MOVJ EC00723
SMOVL C00724 +MOVJ EC00724
SMOVL C00725 +MOVJ EC00725
SMOVL C00726 +MOVJ EC00726
SMOVL C00727 +MOVJ EC00727
SMOVL C00728 +MOVJ EC00728
SMOVL C00729 +MOVJ EC00729
SMOVL C00730 +MOVJ EC00730
SMOVL C00731 +MOVJ EC00731
SMOVL C00732 +MOVJ EC00732
SMOVL C00733 +MOVJ EC00733
SMOVL C00734 +MOVJ EC00734
SMOVL C00735 +MOVJ EC00735
SMOVL C00736 +MOVJ EC00736
SMOVL C00737 +MOVJ EC00737
SMOVL C00738 +MOVJ EC00738
SMOVL C00739 +MOVJ EC00739
SMOVL C00740 +MOVJ EC00740
SMOVL C00741 +MOVJ EC00741
SMOVL C00742 +MOVJ EC00742
SMOVL C00743 +MOVJ EC00743
SMOVL C00744 +MOVJ EC00744
SMOVL C00745 +MOVJ EC00745
SMOVL C00746 +MOVJ EC00746
SMOVL C00747 +MOVJ EC00747
SMOVL C00748 +MOVJ EC00748
SMOVL C00749 +MOVJ EC00749
SMOVL C00750 +MOVJ EC00750
SMOVL C00751 +MOVJ EC00751
SMOVL C00752 +MOVJ EC00752
SMOVL C00753 +MOVJ EC00753
SMOVL C00754 +MOVJ EC00754
SMOVL C00755 +MOVJ EC00755
SMOVL C00756 +MOVJ EC00756
SMOVL C00757 +MOVJ EC00757
SMOVL C00758 +MOVJ EC00758
SMOVL C00759 +MOVJ EC00759
SMOVL C00760 +MOVJ EC00760
SMOVL C00761 +MOVJ EC00761
SMOVL C00762 +MOVJ EC00762
SMOVL C00763 +MOVJ EC00763
SMOVL C00764 +MOVJ EC00764
SMOVL C00765 +MOVJ EC00765
SMOVL C00766 +MOVJ EC00766
SMOVL C00767 +MOVJ EC00767
SMOVL C00768 +MOVJ EC00768
SMOVL C00769 +MOVJ EC00769
SMOVL C00770 +MOVJ EC00770
SMOVL C00771 +MOVJ EC00771
SMOVL C00772 +MOVJ EC00772
SMOVL C00773 +MOVJ EC00773
SMOVL C00774 +MOVJ EC00774
SMOVL C00775 +MOVJ EC00775
SMOVL C00776 +MOVJ EC00776
SMOVL C00777 +MOVJ EC00777
SMOVL C00778 +MOVJ EC00778
SMOVL C00779 +MOVJ EC00779
SMOVL C00780 +MOVJ EC00780
SMOVL C00781 +MOVJ EC00781
SMOVL C00782 +MOVJ EC00782
SMOVL C00783 +MOVJ EC00783
SMOVL C00784 +MOVJ EC00784
SMOVL C00785 +MOVJ EC00785
SMOVL C00786 +MOVJ EC00786
SMOVL C00787 +MOVJ EC00787
SMOVL C00788 +MOVJ EC00788
SMOVL C00789 +MOVJ EC00789
SMOVL C00790 +MOVJ EC00790
SMOVL C00791 +MOVJ EC00791
SMOVL C00792 +MOVJ EC00792
SMOVL C00793 +MOVJ EC00793
SMOVL C00794 +MOVJ EC00794
SMOVL C00795 +MOVJ EC00795
SMOVL C00796 +MOVJ EC00796
SMOVL C00797 +MOVJ EC00797
SMOVL C00798 +MOVJ EC00798
SMOVL C00799 +MOVJ EC00799
SMOVL C00800 +MOVJ EC00800
SMOVL C00801 +MOVJ EC00801
SMOVL C00802 +MOVJ EC00802
SMOVL C00803 +MOVJ EC00803
SMOVL C00804 +MOVJ EC00804
SMOVL C00805 +MOVJ EC00805
SMOVL C00806 +MOVJ EC00806
SMOVL C00807 +MOVJ EC00807
SMOVL C00808 +MOVJ EC00808
SMOVL C00809 +MOVJ EC00809
SMOVL C00810 +MOVJ EC00810
SMOVL C00811 +MOVJ EC00811
SMOVL C00812 +MOVJ EC00812
SMOVL C00813 +MOVJ EC00813
SMOVL C00814 +MOVJ EC00814
SMOVL C00815 +MOVJ EC00815
SMOVL C00816 +MOVJ EC00816
SMOVL C00817 +MOVJ EC00817
SMOVL C00818 +MOVJ EC00818
SMOVL C00819 +MOVJ EC00819
SMOVL C00820 +MOVJ EC00820
SMOVL C00821 +MOVJ EC00821
SMOVL C00822 +MOVJ EC00822
SMOVL C00823 +MOVJ EC00823
SMOVL C00824 +MOVJ EC00824
SMOVL C00825 +MOVJ EC00825
SMOVL C00826 +MOVJ EC00826
SMOVL C00827 +MOVJ EC00827
SMOVL C00828 +MOVJ EC00828
SMOVL C00829 +MOVJ EC00829
SMOVL C00830 +MOVJ EC00830
SMOVL C00831 +MOVJ EC00831
SMOVL C00832 +MOVJ EC00832
SMOVL C00833 +MOVJ EC00833
SMOVL C00834 +MOVJ EC00834
SMOVL C00835 +MOVJ EC00835
SMOVL C00836 +MOVJ EC00836
SMOVL C00837 +MOVJ EC00837
SMOVL C00838 +MOVJ EC00838
SMOVL C00839 +MOVJ EC00839
SMOVL C00840 +MOVJ EC00840
SMOVL C00841 +MOVJ EC00841
SMOVL C00842 +MOVJ EC00842
SMOVL C00843 +MOVJ EC00843
SMOVL C00844 +MOVJ EC00844
SMOVL C00845 +MOVJ EC00845
SMOVL C00846 +MOVJ EC00846
SMOVL C00847 +MOVJ EC00847
SMOVL C00848 +MOVJ EC00848
SMOVL C00849 +MOVJ EC00849
SMOVL C00850 +MOVJ EC00850
SMOVL C00851 +MOVJ EC00851
SMOVL C00852 +MOVJ EC00852
SMOVL C00853 +MOVJ EC00853
SMOVL C00854 +MOVJ EC00854
SMOVL C00855 +MOVJ EC00855
SMOVL C00856 +MOVJ EC00856
SMOVL C00857 +MOVJ EC00857
SMOVL C00858 +MOVJ EC00858
SMOVL C00859 +MOVJ EC00859
SMOVL C00860 +MOVJ EC00860
SMOVL C00861 +MOVJ EC00861
SMOVL C00862 +MOVJ EC00862
SMOVL C00863 +MOVJ EC00863
SMOVL C00864 +MOVJ EC00864
SMOVL C00865 +MOVJ EC00865
SMOVL C00866 +MOVJ EC00866
SMOVL C00867 +MOVJ EC00867
SMOVL C00868 +MOVJ EC00868
SMOVL C00869 +MOVJ EC00869
SMOVL C00870 +MOVJ EC00870
SMOVL C00871 +MOVJ EC00871
SMOVL C00872 +MOVJ EC00872
SMOVL C00873 +MOVJ EC00873
SMOVL C00874 +MOVJ EC00874
SMOVL C00875 +MOVJ EC00875
SMOVL C00876 +MOVJ EC00876
SMOVL C00877 +MOVJ EC00877
SMOVL C00878 +MOVJ EC00878
SMOVL C00879 +MOVJ EC00879
SMOVL C00880 +MOVJ EC00880
SMOVL C00881 +MOVJ EC00881
SMOVL C00882 +MOVJ EC00882
SMOVL C00883 +MOVJ EC00883
SMOVL C00884 +MOVJ EC00884
SMOVL C00885 +MOVJ EC00885
SMOVL C00886 +MOVJ EC00886
SMOVL C00887 +MOVJ EC00887
SMOVL C00888 +MOVJ EC00888
SMOVL C00889 +MOVJ EC00889
SMOVL C00890 +MOVJ EC00890
SMOVL C00891 +MOVJ EC00891
SMOVL C00892 +MOVJ EC00892
SMOVL C00893 +MOVJ EC00893
SMOVL C00894 +MOVJ EC00894
SMOVL C00895 +MOVJ EC00895
SMOVL C00896 +MOVJ EC00896
SMOVL C00897 +MOVJ EC00897
SMOVL C00898 +MOVJ EC00898
SMOVL C00899 +MOVJ EC00899
SMOVL C00900 +MOVJ EC00900
SMOVL C00901 +MOVJ EC00901
SMOVL C00902 +MOVJ EC00902
SMOVL C00903 +MOVJ EC00903
SMOVL C00904 +MOVJ EC00904
SMOVL C00905 +MOVJ EC00905
SMOVL C00906 +MOVJ EC00906
SMOVL C00907 +MOVJ EC00907
SMOVL C00908 +MOVJ EC00908
SMOVL C00909 +MOVJ EC00909
SMOVL C00910 +MOVJ EC00910
SMOVL C00911 +MOVJ EC00911
SMOVL C00912 +MOVJ EC00912
SMOVL C00913 +MOVJ EC00913
SMOVL C00914 +MOVJ EC00914
SMOVL C00915 +MOVJ EC00915
SMOVL C00916 +MOVJ EC00916
SMOVL C00917 +MOVJ EC00917
SMOVL C00918 +MOVJ EC00918
SMOVL C00919 +MOVJ EC00919
SMOVL C00920 +MOVJ EC00920
SMOVL C00921 +MOVJ EC00921
SMOVL C00922 +MOVJ EC00922
SMOVL C00923 +MOVJ EC00923
SMOVL C00924 +MOVJ EC00924
SMOVL C00925 +MOVJ EC00925
SMOVL C00926 +MOVJ EC00926
SMOVL C00927 +MOVJ EC00927
SMOVL C00928 +MOVJ EC00928
SMOVL C00929 +MOVJ EC00929
SMOVL C00930 +MOVJ EC00930
SMOVL C00931 +MOVJ EC00931
SMOVL C00932 +MOVJ EC00932
SMOVL C00933 +MOVJ EC00933
SMOVL C00934 +MOVJ EC00934
SMOVL C00935 +MOVJ EC00935
SMOVL C00936 +MOVJ EC00936
SMOVL C00937 +MOVJ EC00937
SMOVL C00938 +MOVJ EC00938
SMOVL C00939 +MOVJ EC00939
SMOVL C00940 +MOVJ EC00940
SMOVL C00941 +MOVJ EC00941
SMOVL C00942 +MOVJ EC00942
SMOVL C00943 +MOVJ EC00943
SMOVL C00944 +MOVJ EC00944
SMOVL C00945 +MOVJ EC00945
SMOVL C00946 +MOVJ EC00946
SMOVL C00947 +MOVJ EC00947
SMOVL C00948 +MOVJ EC00948
SMOVL C00949 +MOVJ EC00949
SMOVL C00950 +MOVJ EC00950
SMOVL C00951 +MOVJ EC00951
SMOVL C00952 +MOVJ EC00952
SMOVL C00953 +MOVJ EC00953
SMOVL C00954 +MOVJ EC00954
SMOVL C00955 +MOVJ EC00955
SMOVL C00956 +MOVJ EC00956
SMOVL C00957 +MOVJ EC00957
SMOVL C00958 +MOVJ EC00958
SMOVL C00959 +MOVJ EC00959
SMOVL C00960 +MOVJ EC00960
SMOVL C00961 +MOVJ EC00961
SMOVL C00962 +MOVJ EC00962
SMOVL C00963 +MOVJ EC00963
SMOVL C00964 +MOVJ EC00964
SMOVL C00965 +MOVJ EC00965
SMOVL C00966 +MOVJ EC00966
SMOVL C00967 +MOVJ EC00967
SMOVL C00968 +MOVJ EC00968
SMOVL C00969 +MOVJ EC00969
SMOVL C00970 +MOVJ EC00970
SMOVL C00971 +MOVJ EC00971
SMOVL C00972 +MOVJ EC00972
SMOVL C00973 +MOVJ EC00973
SMOVL C00974 +MOVJ EC00974
SMOVL C00975 +MOVJ EC00975
SMOVL C00976 +MOVJ EC00976
SMOVL C00977 +MOVJ EC00977
SMOVL C00978 +MOVJ EC00978
SMOVL C00979 +MOVJ EC00979
SMOVL C00980 +MOVJ EC00980
SMOVL C00981 +MOVJ EC00981
SMOVL C00982 +MOVJ EC00982
SMOVL C00983 +MOVJ EC00983
SMOVL C00984 +MOVJ EC00984
SMOVL C00985 +MOVJ EC00985
SMOVL C00986 +MOVJ EC00986
SMOVL C00987 +MOVJ EC00987
SMOVL C00988 +MOVJ EC00988
SMOVL C00989 +MOVJ EC00989
SMOVL C00990 +MOVJ EC00990
SMOVL C00991 +MOVJ EC00991
SMOVL C00992 +MOVJ EC00992
SMOVL C00993 +MOVJ EC00993
SMOVL C00994 +MOVJ EC00994
SMOVL C00995 +MOVJ EC00995
SMOVL C00996 +MOVJ EC00996
SMOVL C00997 +MOVJ EC00997
SMOVL C00998 +MOVJ EC00998
SMOVL C00999 +MOVJ EC00999
SMOVL C01000 +MOVJ EC01000
SMOVL C01001 +MOVJ EC01001
SMOVL C01002 +MOVJ EC01002
SMOVL C01003 +MOVJ EC01003
SMOVL C01004 +MOVJ EC01004
SMOVL C01005 +MOVJ EC01005
SMOVL C01006 +MOVJ EC01006
SMOVL C01007 +MOVJ EC01007
SMOVL C01008 +MOVJ EC01008
SMOVL C01009 +MOVJ EC01009
SMOVL C01010 +MOVJ EC01010
SMOVL C01011 +MOVJ EC01011
SMOVL C01012 +MOVJ EC01012
SMOVL C01013 +MOVJ EC01013
SMOVL C01014 +MOVJ EC01014
SMOVL C01015 +MOVJ EC01015
SMOVL C01016 +MOVJ EC01016
SMOVL C01017 +MOVJ EC01017
SMOVL C01018 +MOVJ EC01018
SMOVL C01019 +MOVJ EC01019
SMOVL C01020 +MOVJ EC01020
SMOVL C01021 +MOVJ EC01021
SMOVL C01022 +MOVJ EC01022
SMOVL C01023 +MOVJ EC01023
SMOVL C01024 +MOVJ EC01024
SMOVL C01025 +MOVJ EC01025
SMOVL C01026 +MOVJ EC01026
SMOVL C01027 +MOVJ EC01027
SMOVL C01028 +MOVJ EC01028
SMOVL C01029 +MOVJ EC01029
SMOVL C01030 +MOVJ EC01030
SMOVL C01031 +MOVJ EC01031
SMOVL C01032 +MOVJ EC01032
SMOVL C01033 +MOVJ EC01033
SMOVL C01034 +MOVJ EC01034
SMOVL C01035 +MOVJ EC01035
SMOVL C01036 +MOVJ EC01036
SMOVL C01037 +MOVJ EC01037
SMOVL C01038 +MOVJ EC01038
SMOVL C01039 +MOVJ EC01039
SMOVL C01040 +MOVJ EC01040
SMOVL C01041 +MOVJ EC01041
SMOVL C01042 +MOVJ EC01042
SMOVL C01043 +MOVJ EC01043
SMOVL C01044 +MOVJ EC01044
SMOVL C01045 +MOVJ EC01045
SMOVL C01046 +MOVJ EC01046
SMOVL C01047 +MOVJ EC01047
SMOVL C01048 +MOVJ EC01048
SMOVL C01049 +MOVJ EC01049
SMOVL C01050 +MOVJ EC01050
SMOVL C01051 +MOVJ EC01051
SMOVL C01052 +MOVJ EC01052
SMOVL C01053 +MOVJ EC01053
SMOVL C01054 +MOVJ EC01054
SMOVL C01055 +MOVJ EC01055
SMOVL C01056 +MOVJ EC01056
SMOVL C01057 +MOVJ EC01057
SMOVL C01058 +MOVJ EC01058
SMOVL C01059 +MOVJ EC01059
SMOVL C01060 +MOVJ EC01060
SMOVL C01061 +MOVJ EC01061
SMOVL C01062 +MOVJ EC01062
SMOVL C01063 +MOVJ EC01063
SMOVL C01064 +MOVJ EC01064
SMOVL C01065 +MOVJ EC01065
SMOVL C01066 +MOVJ EC01066
SMOVL C01067 +MOVJ EC01067
SMOVL C01068 +MOVJ EC01068
SMOVL C01069 +MOVJ EC01069
SMOVL C01070 +MOVJ EC01070
SMOVL C01071 +MOVJ EC01071
SMOVL C01072 +MOVJ EC01072
SMOVL C01073 +MOVJ EC01073
SMOVL C01074 +MOVJ EC01074
SMOVL C01075 +MOVJ EC01075
SMOVL C01076 +MOVJ EC01076
SMOVL C01077 +MOVJ EC01077
SMOVL C01078 +MOVJ EC01078
SMOVL C01079 +MOVJ EC01079
SMOVL C01080 +MOVJ EC01080
SMOVL C01081 +MOVJ EC01081
SMOVL C01082 +MOVJ EC01082
SMOVL C01083 +MOVJ EC01083
SMOVL C01084 +MOVJ EC01084
SMOVL C01085 +MOVJ EC01085
SMOVL C01086 +MOVJ EC01086
SMOVL C01087 +MOVJ EC01087
SMOVL C01088 +MOVJ EC01088
SMOVL C01089 +MOVJ EC01089
SMOVL C01090 +MOVJ EC01090
SMOVL C01091 +MOVJ EC01091
SMOVL C01092 +MOVJ EC01092
SMOVL C01093 +MOVJ EC01093
SMOVL C01094 +MOVJ EC01094
SMOVL C01095 +MOVJ EC01095
SMOVL C01096 +MOVJ EC01096
SMOVL C01097 +MOVJ EC01097
SMOVL C01098 +MOVJ EC01098
SMOVL C01099 +MOVJ EC01099
SMOVL C01100 +MOVJ EC01100
SMOVL C01101 +MOVJ EC01101
SMOVL C01102 +MOVJ EC01102
SMOVL C01103 +MOVJ EC01103
SMOVL C01104 +MOVJ EC01104
SMOVL C01105 +MOVJ EC01105
SMOVL C01106 +MOVJ EC01106
SMOVL C01107 +MOVJ EC01107
SMOVL C01108 +MOVJ EC01108
SMOVL C01109 +MOVJ EC01109
SMOVL C01110 +MOVJ EC01110
SMOVL C01111 +MOVJ EC01111
SMOVL C01112 +MOVJ EC01112
SMOVL C01113 +MOVJ EC01113
SMOVL C01114 +MOVJ EC01114
SMOVL C01115 +MOVJ EC01115
SMOVL C01116 +MOVJ EC01116
SMOVL C01117 +MOVJ EC01117
SMOVL C01118 +MOVJ EC01118
SMOVL C01119 +MOVJ EC01119
SMOVL C01120 +MOVJ EC01120
SMOVL C01121 +MOVJ EC01121
SMOVL C01122 +MOVJ EC01122
SMOVL C01123 +MOVJ EC01123
SMOVL C01124 +MOVJ EC01124
SMOVL C01125 +MOVJ EC01125
SMOVL C01126 +MOVJ EC01126
SMOVL C01127 +MOVJ EC01127
SMOVL C01128 +MOVJ EC01128
SMOVL C01129 +MOVJ EC01129
SMOVL C01130 +MOVJ EC01130
SMOVL C01131 +MOVJ EC01131
SMOVL C01132 +MOVJ EC01132
SMOVL C01133 +MOVJ EC01133
SMOVL C01134 +MOVJ EC01134
SMOVL C01135 +MOVJ EC01135
SMOVL C01136 +MOVJ EC01136
SMOVL C01137 +MOVJ EC01137
SMOVL C01138 +MOVJ EC01138
SMOVL C01139 +MOVJ EC01139
SMOVL C01140 +MOVJ EC01140
SMOVL C01141 +MOVJ EC01141
SMOVL C01142 +MOVJ EC01142
SMOVL C01143 +MOVJ EC01143
SMOVL C01144 +MOVJ EC01144
SMOVL C01145 +MOVJ EC01145
SMOVL C01146 +MOVJ EC01146
SMOVL C01147 +MOVJ EC01147
SMOVL C01148 +MOVJ EC01148
SMOVL C01149 +MOVJ EC01149
SMOVL C01150 +MOVJ EC01150
SMOVL C01151 +MOVJ EC01151
SMOVL C01152 +MOVJ EC01152
SMOVL C01153 +MOVJ EC01153
SMOVL C01154 +MOVJ EC01154
SMOVL C01155 +MOVJ EC01155
SMOVL C01156 +MOVJ EC01156
SMOVL C01157 +MOVJ EC01157
SMOVL C01158 +MOVJ EC01158
SMOVL C01159 +MOVJ EC01159
SMOVL C01160 +MOVJ EC01160
SMOVL C01161 +MOVJ EC01161
SMOVL C01162 +MOVJ EC01162
SMOVL C01163 +MOVJ EC01163
SMOVL C01164 +MOVJ EC01164
SMOVL C01165 +MOVJ EC01165
SMOVL C01166 +MOVJ EC01166
SMOVL C01167 +MOVJ EC01167
SMOVL C01168 +MOVJ EC01168
SMOVL C01169 +MOVJ EC01169
SMOVL C01170 +MOVJ EC01170
SMOVL C01171 +MOVJ EC01171
SMOVL C01172 +MOVJ EC01172
SMOVL C01173 +MOVJ EC01173
SMOVL C01174 +MOVJ EC01174
SMOVL C01175 +MOVJ EC01175
SMOVL C01176 +MOVJ EC01176
SMOVL C01177 +MOVJ EC01177
SMOVL C01178 +MOVJ EC01178
SMOVL C01179 +MOVJ EC01179
SMOVL C01180 +MOVJ EC01180
SMOVL C01181 +MOVJ EC01181
SMOVL C01182 +MOVJ EC01182
SMOVL C01183 +MOVJ EC01183
SMOVL C01184 +MOVJ EC01184
SMOVL C01185 +MOVJ EC01185
SMOVL C01186 +MOVJ EC01186
SMOVL C01187 +MOVJ EC01187
SMOVL C01188 +MOVJ EC01188
SMOVL C01189 +MOVJ EC01189
SMOVL C01190 +MOVJ EC01190
SMOVL C01191 +MOVJ EC01191
SMOVL C01192 +MOVJ EC01192
SMOVL C01193 +MOVJ EC01193
SMOVL C01194 +MOVJ EC01194
SMOVL C01195 +MOVJ EC01195
SMOVL C01196 +MOVJ EC01196
SMOVL C01197 +MOVJ EC01197
SMOVL C01198 +MOVJ EC01198
SMOVL C01199 +MOVJ EC01199
SMOVL C01200 +MOVJ EC01200
SMOVL C01201 +MOVJ EC01201
SMOVL C01202 +MOVJ EC01202
SMOVL C01203 +MOVJ EC01203
SMOVL C01204 +MOVJ EC01204
SMOVL C01205 +MOVJ EC01205
SMOVL C01206 +MOVJ EC01206
SMOVL C01207 +MOVJ EC01207
SMOVL C01208 +MOVJ EC01208
SMOVL C01209 +MOVJ EC01209
SMOVL C01210 +MOVJ EC01210
SMOVL C01211 +MOVJ EC01211
SMOVL C01212 +MOVJ EC01212
SMOVL C01213 +MOVJ EC01213
SMOVL C01214 +MOVJ EC01214
SMOVL C01215 +MOVJ EC01215
SMOVL C01216 +MOVJ EC01216
SMOVL C01217 +MOVJ EC01217
SMOVL C01218 +MOVJ EC01218
SMOVL C01219 +MOVJ EC01219
SMOVL C01220 +MOVJ EC01220
SMOVL C01221 +MOVJ EC01221
SMOVL C01222 +MOVJ EC01222
SMOVL C01223 +MOVJ EC01223
SMOVL C01224 +MOVJ EC01224
SMOVL C01225 +MOVJ EC01225
SMOVL C01226 +MOVJ EC01226
SMOVL C01227 +MOVJ EC01227
SMOVL C01228 +MOVJ EC01228
SMOVL C01229 +MOVJ EC01229
SMOVL C01230 +MOVJ EC01230
SMOVL C01231 +MOVJ EC01231
SMOVL C01232 +MOVJ EC01232
SMOVL C01233 +MOVJ EC01233
SMOVL C01234 +MOVJ EC01234
SMOVL C01235 +MOVJ EC01235
SMOVL C01236 +MOVJ EC01236
SMOVL C01237 +MOVJ EC01237
SMOVL C01238 +MOVJ EC01238
SMOVL C01239 +MOVJ EC01239
SMOVL C01240 +MOVJ EC01240
SMOVL C01241 +MOVJ EC01241
SMOVL C01242 +MOVJ EC01242
SMOVL C01243 +MOVJ EC01243
SMOVL C01244 +MOVJ EC01244
SMOVL C01245 +MOVJ EC01245
SMOVL C01246 +MOVJ EC01246
SMOVL C01247 +MOVJ EC01247
SMOVL C01248 +MOVJ EC01248
SMOVL C01249 +MOVJ EC01249
SMOVL C01250 +MOVJ EC01250
SMOVL C01251 +MOVJ EC01251
SMOVL C01252 +MOVJ EC01252
SMOVL C01253 +MOVJ EC01253
SMOVL C01254 +MOVJ EC01254
SMOVL C01255 +MOVJ EC01255
SMOVL C01256 +MOVJ EC01256
SMOVL C01257 +MOVJ EC01257
SMOVL C01258 +MOVJ EC01258
SMOVL C01259 +MOVJ EC01259
SMOVL C01260 +MOVJ EC01260
SMOVL C01261 +MOVJ EC01261
SMOVL C01262 +MOVJ EC01262
SMOVL C01263 +MOVJ EC01263
SMOVL C01264 +MOVJ EC01264
SMOVL C01265 +MOVJ EC01265
SMOVL C01266 +MOVJ EC01266
SMOVL C01267 +MOVJ EC01267
SMOVL C01268 +MOVJ EC01268
SMOVL C01269 +MOVJ EC01269
SMOVL C01270 +MOVJ EC01270
SMOVL C01271 +MOVJ EC01271
SMOVL C01272 +MOVJ EC01272
SMOVL C01273 +MOVJ EC01273
SMOVL C01274 +MOVJ EC01274
SMOVL C01275 +MOVJ EC01275
SMOVL C01276 +MOVJ EC01276
SMOVL C01277 +MOVJ EC01277
SMOVL C01278 +MOVJ EC01278
SMOVL C01279 +MOVJ EC01279
SMOVL C01280 +MOVJ EC01280
SMOVL C01281 +MOVJ EC01281
SMOVL C01282 +MOVJ EC01282
SMOVL C01283 +MOVJ EC01283
SMOVL C01284 +MOVJ EC01284
SMOVL C01285 +MOVJ EC01285
SMOVL C01286 +MOVJ EC01286
SMOVL C01287 +MOVJ EC01287
SMOVL C01288 +MOVJ EC01288
SMOVL C01289 +MOVJ EC01289
SMOVL C01290 +MOVJ EC01290
SMOVL C01291 +MOVJ EC01291
SMOVL C01292 +MOVJ EC01292
SMOVL C01293 +MOVJ EC01293
SMOVL C01294 +MOVJ EC01294
SMOVL C01295 +MOVJ EC01295
SMOVL C01296 +MOVJ EC01296
SMOVL C01297 +MOVJ EC01297
SMOVL C01298 +MOVJ EC01298
SMOVL C01299 +MOVJ EC01299
SMOVL C01300 +MOVJ EC01300
SMOVL C01301 +MOVJ EC01301
SMOVL C01302 +MOVJ EC01302
SMOVL C01303 +MOVJ EC01303
SMOVL C01304 +MOVJ EC01304
SMOVL C01305 +MOVJ EC01305
SMOVL C01306 +MOVJ EC01306
SMOVL C01307 +MOVJ EC01307
SMOVL C01308 +MOVJ EC01308
SMOVL C01309 +MOVJ EC01309
SMOVL C01310 +MOVJ EC01310
SMOVL C01311 +MOVJ EC01311
SMOVL C01312 +MOVJ EC01312
SMOVL C01313 +MOVJ EC01313
SMOVL C01314 +MOVJ EC01314
SMOVL C01315 +MOVJ EC01315
SMOVL C01316 +MOVJ EC01316
SMOVL C01317 +MOVJ EC01317
SMOVL C01318 +MOVJ EC01318
SMOVL C01319 +MOVJ EC01319
SMOVL C01320 +MOVJ EC01320
SMOVL C01321 +MOVJ EC01321
SMOVL C01322 +MOVJ EC01322
SMOVL C01323 +MOVJ EC01323
SMOVL C01324 +MOVJ EC01324
SMOVL C01325 +MOVJ EC01325
SMOVL C01326 +MOVJ EC01326
SMOVL C01327 +MOVJ EC01327
SMOVL C01328 +MOVJ EC01328
SMOVL C01329 +MOVJ EC01329
SMOVL C01330 +MOVJ EC01330
SMOVL C01331 +MOVJ EC01331
SMOVL C01332 +MOVJ EC01332
SMOVL C01333 +MOVJ EC01333
SMOVL C01334 +MOVJ EC01334
SMOVL C01335 +MOVJ EC01335
SMOVL C01336 +MOVJ EC01336
SMOVL C01337 +MOVJ EC01337
SMOVL C01338 +MOVJ EC01338
SMOVL C01339 +MOVJ EC01339
SMOVL C01340 +MOVJ EC01340
SMOVL C01341 +MOVJ EC01341
SMOVL C01342 +MOVJ EC01342
SMOVL C01343 +MOVJ EC01343
SMOVL C01344 +MOVJ EC01344
SMOVL C01345 +MOVJ EC01345
SMOVL C01346 +MOVJ EC01346
SMOVL C01347 +MOVJ EC01347
SMOVL C01348 +MOVJ EC01348
SMOVL C01349 +MOVJ EC01349
SMOVL C01350 +MOVJ EC01350
SMOVL C01351 +MOVJ EC01351
SMOVL C01352 +MOVJ EC01352
SMOVL C01353 +MOVJ EC01353
SMOVL C01354 +MOVJ EC01354
SMOVL C01355 +MOVJ EC01355
SMOVL C01356 +MOVJ EC01356
SMOVL C01357 +MOVJ EC01357
SMOVL C01358 +MOVJ EC01358
SMOVL C01359 +MOVJ EC01359
SMOVL C01360 +MOVJ EC01360
SMOVL C01361 +MOVJ EC01361
SMOVL C01362 +MOVJ EC01362
SMOVL C01363 +MOVJ EC01363
SMOVL C01364 +MOVJ EC01364
SMOVL C01365 +MOVJ EC01365
SMOVL C01366 +MOVJ EC01366
SMOVL C01367 +MOVJ EC01367
SMOVL C01368 +MOVJ EC01368
SMOVL C01369 +MOVJ EC01369
SMOVL C01370 +MOVJ EC01370
SMOVL C01371 +MOVJ EC01371
SMOVL C01372 +MOVJ EC01372
SMOVL C01373 +MOVJ EC01373
SMOVL C01374 +MOVJ EC01374
SMOVL C01375 +MOVJ EC01375
SMOVL C01376 +MOVJ EC01376
SMOVL C01377 +MOVJ EC01377
SMOVL C01378 +MOVJ EC01378
SMOVL C01379 +MOVJ EC01379
SMOVL C01380 +MOVJ EC01380
SMOVL C01381 +MOVJ EC01381
SMOVL C01382 +MOVJ EC01382
SMOVL C01383 +MOVJ EC01383
SMOVL C01384 +MOVJ EC01384
SMOVL C01385 +MOVJ EC01385
SMOVL C01386 +MOVJ EC01386
SMOVL C01387 +MOVJ EC01387
SMOVL C01388 +MOVJ EC01388
SMOVL C01389 +MOVJ EC01389
SMOVL C01390 +MOVJ EC01390
SMOVL C01391 +MOVJ EC01391
SMOVL C01392 +MOVJ EC01392
SMOVL C01393 +MOVJ EC01393
SMOVL C01394 +MOVJ EC01394
SMOVL C01395 +MOVJ EC01395
SMOVL C01396 +MOVJ EC01396
SMOVL C01397 +MOVJ EC01397
SMOVL C01398 +MOVJ EC01398
SMOVL C01399 +MOVJ EC01399
SMOVL C01400 +MOVJ EC01400
SMOVL C01401 +MOVJ EC01401
SMOVL C01402 +MOVJ EC01402
SMOVL C01403 +MOVJ EC01403
SMOVL C01404 +MOVJ EC01404
SMOVL C01405 +MOVJ EC01405
SMOVL C01406 +MOVJ EC01406
SMOVL C01407 +MOVJ EC01407
SMOVL C01408 +MOVJ EC01408
SMOVL C01409 +MOVJ EC01409
SMOVL C01410 +MOVJ EC01410
SMOVL C01411 +MOVJ EC01411
SMOVL C01412 +MOVJ EC01412
SMOVL C01413 +MOVJ EC01413
SMOVL C01414 +MOVJ EC01414
SMOVL C01415 +MOVJ EC01415
SMOVL C01416 +MOVJ EC01416
SMOVL C01417 +MOVJ EC01417
SMOVL C01418 +MOVJ EC01418
SMOVL C01419 +MOVJ EC01419
SMOVL C01420 +MOVJ EC01420
SMOVL C01421 +MOVJ EC01421
SMOVL C01422 +MOVJ EC01422
SMOVL C01423 +MOVJ EC01423
SMOVL C01424 +MOVJ EC01424
SMOVL C01425 +MOVJ EC01425
SMOVL C01426 +MOVJ EC01426
SMOVL C01427 +MOVJ EC01427
SMOVL C01428 +MOVJ EC01428
SMOVL C01429 +MOVJ EC01429
SMOVL C01430 +MOVJ EC01430
SMOVL C01431 +MOVJ EC01431
SMOVL C01432 +MOVJ EC01432
SMOVL C01433 +MOVJ EC01433
SMOVL C01434 +MOVJ EC01434
SMOVL C01435 +MOVJ EC01435
SMOVL C01436 +MOVJ EC01436
SMOVL C01437 +MOVJ EC01437
SMOVL C01438 +MOVJ EC01438
SMOVL C01439 +MOVJ EC01439
SMOVL C01440 +MOVJ EC01440
SMOVL C01441 +MOVJ EC01441
SMOVL C01442 +MOVJ EC01442
SMOVL C01443 +MOVJ EC01443
SMOVL C01444 +MOVJ EC01444
SMOVL C01445 +MOVJ EC01445
SMOVL C01446 +MOVJ EC01446
SMOVL C01447 +MOVJ EC01447
SMOVL C01448 +MOVJ EC01448
SMOVL C01449 +MOVJ EC01449
SMOVL C01450 +MOVJ EC01450
SMOVL C01451 +MOVJ EC01451
SMOVL C01452 +MOVJ EC01452
SMOVL C01453 +MOVJ EC01453
SMOVL C01454 +MOVJ EC01454
SMOVL C01455 +MOVJ EC01455
SMOVL C01456 +MOVJ EC01456
SMOVL C01457 +MOVJ EC01457
SMOVL C01458 +MOVJ EC01458
SMOVL C01459 +MOVJ EC01459
SMOVL C01460 +MOVJ EC01460
SMOVL C01461 +MOVJ EC01461
SMOVL C01462 +MOVJ EC01462
SMOVL C01463 +MOVJ EC01463
SMOVL C01464 +MOVJ EC01464
SMOVL C01465 +MOVJ EC01465
SMOVL C01466 +MOVJ EC01466
SMOVL C01467 +MOVJ EC01467
SMOVL C01468 +MOVJ EC01468
SMOVL C01469 +MOVJ EC01469
SMOVL C01470 +MOVJ EC01470
SMOVL C01471 +MOVJ EC01471
SMOVL C01472 +MOVJ EC01472
SMOVL C01473 +MOVJ EC01473
SMOVL C01474 +MOVJ EC01474
SMOVL C01475 +MOVJ EC01475
SMOVL C01476 +MOVJ EC01476
SMOVL C01477 +MOVJ EC01477
SMOVL C01478 +MOVJ EC01478
SMOVL C01479 +MOVJ EC01479
SMOVL C01480 +MOVJ EC01480
SMOVL C01481 +MOVJ EC01481
SMOVL C01482 +MOVJ EC01482
SMOVL C01483 +MOVJ EC01483
SMOVL C01484 +MOVJ EC01484
SMOVL C01485 +MOVJ EC01485
SMOVL C01486 +MOVJ EC01486
SMOVL C01487 +MOVJ EC01487
SMOVL C01488 +MOVJ EC01488
SMOVL C01489 +MOVJ EC01489
SMOVL C01490 +MOVJ EC01490
SMOVL C01491 +MOVJ EC01491
SMOVL C01492 +MOVJ EC01492
SMOVL C01493 +MOVJ EC01493
SMOVL C01494 +MOVJ EC01494
SMOVL C01495 +MOVJ EC01495
SMOVL C01496 +MOVJ EC01496
SMOVL C01497 +MOVJ EC01497
SMOVL C01498 +MOVJ EC01498
SMOVL C01499 +MOVJ EC01499
SMOVL C01500 +MOVJ EC01500
SMOVL C01501 +MOVJ EC01501
SMOVL C01502 +MOVJ EC01502
SMOVL C01503 +MOVJ EC01503
SMOVL C01504 +MOVJ EC01504
SMOVL C01505 +MOVJ EC01505
SMOVL C01506 +MOVJ EC01506
SMOVL C01507 +MOVJ EC01507
SMOVL C01508 +MOVJ EC01508
SMOVL C01509 +MOVJ EC01509
SMOVL C01510 +MOVJ EC01510
SMOVL C01511 +MOVJ EC01511
SMOVL C01512 +MOVJ EC01512
SMOVL C01513 +MOVJ EC01513
SMOVL C01514 +MOVJ EC01514
SMOVL C01515 +MOVJ EC01515
SMOVL C01516 +MOVJ EC01516
SMOVL C01517 +MOVJ EC01517
SMOVL C01518 +MOVJ EC01518
SMOVL C01519 +MOVJ EC01519
SMOVL C01520 +MOVJ EC01520
SMOVL C01521 +MOVJ EC01521
SMOVL C01522 +MOVJ EC01522
SMOVL C01523 +MOVJ EC01523
SMOVL C01524 +MOVJ EC01524
SMOVL C01525 +MOVJ EC01525
SMOVL C01526 +MOVJ EC01526
SMOVL C01527 +MOVJ EC01527
SMOVL C01528 +MOVJ EC01528
SMOVL C01529 +MOVJ EC01529
SMOVL C01530 +MOVJ EC01530
SMOVL C01531 +MOVJ EC01531
SMOVL C01532 +MOVJ EC01532
SMOVL C01533 +MOVJ EC01533
SMOVL C01534 +MOVJ EC01534
SMOVL C01535 +MOVJ EC01535
SMOVL C01536 +MOVJ EC01536
SMOVL C01537 +MOVJ EC01537
SMOVL C01538 +MOVJ EC01538
SMOVL C01539 +MOVJ EC01539
SMOVL C01540 +MOVJ EC01540
SMOVL C01541 +MOVJ EC01541
SMOVL C01542 +MOVJ EC01542
SMOVL C01543 +MOVJ EC01543
SMOVL C01544 +MOVJ EC01544
SMOVL C01545 +MOVJ EC01545
SMOVL C01546 +MOVJ EC01546
SMOVL C01547 +MOVJ EC01547
SMOVL C01548 +MOVJ EC01548
SMOVL C01549 +MOVJ EC01549
SMOVL C01550 +MOVJ EC01550
SMOVL C01551 +MOVJ EC01551
SMOVL C01552 +MOVJ EC01552
SMOVL C01553 +MOVJ EC01553
SMOVL C01554 +MOVJ EC01554
SMOVL C01555 +MOVJ EC01555
SMOVL C01556 +MOVJ EC01556
SMOVL C01557 +MOVJ EC01557
SMOVL C01558 +MOVJ EC01558
SMOVL C01559 +MOVJ EC01559
SMOVL C01560 +MOVJ EC01560
SMOVL C01561 +MOVJ EC01561
SMOVL C01562 +MOVJ EC01562
SMOVL C01563 +MOVJ EC01563
SMOVL C01564 +MOVJ EC01564
SMOVL C01565 +MOVJ EC01565
SMOVL C01566 +MOVJ EC01566
SMOVL C01567 +MOVJ EC01567
SMOVL C01568 +MOVJ EC01568
SMOVL C01569 +MOVJ EC01569
SMOVL C01570 +MOVJ EC01570
SMOVL C01571 +MOVJ EC01571
SMOVL C01572 +MOVJ EC01572
SMOVL C01573 +MOVJ EC01573
SMOVL C01574 +MOVJ EC01574
SMOVL C01575 +MOVJ EC01575
SMOVL C01576 +MOVJ EC01576
SMOVL C01577 +MOVJ EC01577
SMOVL C01578 +MOVJ EC01578
SMOVL C01579 +MOVJ EC01579
SMOVL C01580 +MOVJ EC01580
SMOVL C01581 +MOVJ EC01581
SMOVL C01582 +MOVJ EC01582
SMOVL C01583 +MOVJ EC01583
SMOVL C01584 +MOVJ EC01584
SMOVL C01585 +MOVJ EC01585
SMOVL C01586 +MOVJ EC01586
SMOVL C01587 +MOVJ EC01587
SMOVL C01588 +MOVJ EC01588
SMOVL C01589 +MOVJ EC01589
SMOVL C01590 +MOVJ EC01590
SMOVL C01591 +MOVJ EC01591
SMOVL C01592 +MOVJ EC01592
SMOVL C01593 +MOVJ EC01593
SMOVL C01594 +MOVJ EC01594
SMOVL C01595 +MOVJ EC01595
SMOVL C01596 +MOVJ EC01596
SMOVL C01597 +MOVJ EC01597
SMOVL C01598 +MOVJ EC01598
SMOVL C01599 +MOVJ EC01599
SMOVL C01600 +MOVJ EC01600
SMOVL C01601 +MOVJ EC01601
SMOVL C01602 +MOVJ EC01602
SMOVL C01603 +MOVJ EC01603
SMOVL C01604 +MOVJ EC01604
SMOVL C01605 +MOVJ EC01605
SMOVL C01606 +MOVJ EC01606
SMOVL C01607 +MOVJ EC01607
SMOVL C01608 +MOVJ EC01608
SMOVL C01609 +MOVJ EC01609
SMOVL C01610 +MOVJ EC01610
SMOVL C01611 +MOVJ EC01611
SMOVL C01612 +MOVJ EC01612
SMOVL C01613 +MOVJ EC01613
SMOVL C01614 +MOVJ EC01614
SMOVL C01615 +MOVJ EC01615
SMOVL C01616 +MOVJ EC01616
SMOVL C01617 +MOVJ EC01617
SMOVL C01618 +MOVJ EC01618
SMOVL C01619 +MOVJ EC01619
SMOVL C01620 +MOVJ EC01620
SMOVL C01621 +MOVJ EC01621
SMOVL C01622 +MOVJ EC01622
SMOVL C01623 +MOVJ EC01623
SMOVL C01624 +MOVJ EC01624
SMOVL C01625 +MOVJ EC01625
SMOVL C01626 +MOVJ EC01626
SMOVL C01627 +MOVJ EC01627
SMOVL C01628 +MOVJ EC01628
SMOVL C01629 +MOVJ EC01629
SMOVL C01630 +MOVJ EC01630
SMOVL C01631 +MOVJ EC01631
SMOVL C01632 +MOVJ EC01632
SMOVL C01633 +MOVJ EC01633
SMOVL C01634 +MOVJ EC01634
SMOVL C01635 +MOVJ EC01635
SMOVL C01636 +MOVJ EC01636
SMOVL C01637 +MOVJ EC01637
SMOVL C01638 +MOVJ EC01638
SMOVL C01639 +MOVJ EC01639
SMOVL C01640 +MOVJ EC01640
SMOVL C01641 +MOVJ EC01641
SMOVL C01642 +MOVJ EC01642
SMOVL C01643 +MOVJ EC01643
SMOVL C01644 +MOVJ EC01644
SMOVL C01645 +MOVJ EC01645
SMOVL C01646 +MOVJ EC01646
SMOVL C01647 +MOVJ EC01647
SMOVL C01648 +MOVJ EC01648
SMOVL C01649 +MOVJ EC01649
SMOVL C01650 +MOVJ EC01650
SMOVL C01651 +MOVJ EC01651
SMOVL C01652 +MOVJ EC01652
SMOVL C01653 +MOVJ EC01653
SMOVL C01654 +MOVJ EC01654
SMOVL C01655 +MOVJ EC01655
SMOVL C01656 +MOVJ EC01656
SMOVL C01657 +MOVJ EC01657
SMOVL C01658 +MOVJ EC01658
SMOVL C01659 +MOVJ EC01659
SMOVL C01660 +MOVJ EC01660
SMOVL C01661 +MOVJ EC01661
SMOVL C01662 +MOVJ EC01662
SMOVL C01663 +MOVJ EC01663
SMOVL C01664 +MOVJ EC01664
SMOVL C01665 +MOVJ EC01665
SMOVL C01666 +MOVJ EC01666
SMOVL C01667 +MOVJ EC01667
SMOVL C01668 +MOVJ EC01668
SMOVL C01669 +MOVJ EC01669
SMOVL C01670 +MOVJ EC01670
SMOVL C01671 +MOVJ EC01671
SMOVL C01672 +MOVJ EC01672
SMOVL C01673 +MOVJ EC01673
SMOVL C01674 +MOVJ EC01674
SMOVL C01675 +MOVJ EC01675
SMOVL C01676 +MOVJ EC01676
SMOVL C01677 +MOVJ EC01677
SMOVL C01678 +MOVJ EC01678
SMOVL C01679 +MOVJ EC01679
SMOVL C01680 +MOVJ EC01680
SMOVL C01681 +MOVJ EC01681
SMOVL C01682 +MOVJ EC01682
SMOVL C01683 +MOVJ EC01683
SMOVL C01684 +MOVJ EC01684
SMOVL C01685 +MOVJ EC01685
SMOVL C01686 +MOVJ EC01686
SMOVL C01687 +MOVJ EC01687
SMOVL C01688 +MOVJ EC01688
SMOVL C01689 +MOVJ EC01689
SMOVL C01690 +MOVJ EC01690
SMOVL C01691 +MOVJ EC01691
SMOVL C01692 +MOVJ EC01692
SMOVL C01693 +MOVJ EC01693
SMOVL C01694 +MOVJ EC01694
SMOVL C01695 +MOVJ EC01695
SMOVL C01696 +MOVJ EC01696
SMOVL C01697 +MOVJ EC01697
SMOVL C01698 +MOVJ EC01698
SMOVL C01699 +MOVJ EC01699
SMOVL C01700 +MOVJ EC01700
SMOVL C01701 +MOVJ EC01701
SMOVL C01702 +MOVJ EC01702
SMOVL C01703 +MOVJ EC01703
SMOVL C01704 +MOVJ EC01704
SMOVL C01705 +MOVJ EC01705
SMOVL C01706 +MOVJ EC01706
SMOVL C01707 +MOVJ EC01707
SMOVL C01708 +MOVJ EC01708
SMOVL C01709 +MOVJ EC01709
SMOVL C01710 +MOVJ EC01710
SMOVL C01711 +MOVJ EC01711
